DATA_BLOCK "Working_Programs"   // DB25
{ S7_Optimized_Access := 'FALSE' }
VERSION : 0.1
   VAR
      Count : USInt := 16;
      List : Array[0..21] of "RobotProgram";
   END_VAR
BEGIN
   List[4].Entry_Points[7].part_side := '';
   List[4].Entry_Points[7].operation_side := '';
   List[4].Entry_Points[7].lay_number := -1;
   List[4].Entry_Points[7].operation_type := 'transfer_slot2out';
   List[4].Entry_Points[7].part_destination := '';
   List[4].Entry_Points[7].part_status := 'gripper';
   List[4].Entry_Points[7].robot_status := 'home';
   List[4].Entry_Points[7].machine_status := '';
   List[4].Entry_Points[7].previous_trajectory := 'TakeFromSlot';
   List[4].Entry_Points[7].active := true;
   List[3].Entry_Points[3].part_side := '';
   List[3].Entry_Points[3].operation_side := '';
   List[3].Entry_Points[3].lay_number := -1;
   List[3].Entry_Points[3].operation_type := 'transfer_in2slot';
   List[3].Entry_Points[3].part_destination := 'part_slot';
   List[3].Entry_Points[3].part_status := 'gripper';
   List[3].Entry_Points[3].robot_status := 'pallet_in';
   List[3].Entry_Points[3].machine_status := '';
   List[3].Entry_Points[3].previous_trajectory := 'TakeFromPalletIn';
   List[3].Entry_Points[3].active := true;
   List[2].Entry_Points[1].operation_type := 'machining';
   List[2].Entry_Points[1].lay_number := -1;
   List[2].Entry_Points[1].operation_side := 'B';
   List[2].Entry_Points[1].part_side := 'B';
   List[2].Entry_Points[2].active := true;
   List[2].Entry_Points[2].previous_trajectory := 'AutoMachiningA_';
   List[2].Entry_Points[2].machine_status := '';
   List[2].Entry_Points[2].robot_status := 'flip_table';
   List[2].Entry_Points[2].part_status := 'flip_table';
   List[2].Entry_Points[2].part_destination := 'pallet_out';
   List[2].Entry_Points[2].operation_type := 'machining';
   List[2].Entry_Points[2].lay_number := -1;
   List[2].Entry_Points[2].operation_side := 'B';
   List[2].Entry_Points[2].part_side := 'B';
   List[15].Entry_Points[1].active := true;
   List[15].Entry_Points[1].previous_trajectory := 'Pallet_Scanning';
   List[15].Entry_Points[1].machine_status := '';
   List[15].Entry_Points[1].robot_status := 'home';
   List[15].Entry_Points[1].part_status := 'pallet_in';
   List[15].Entry_Points[1].part_destination := 'pallet_out';
   List[6].Entry_Points[9].part_side := 'A';
   List[6].Entry_Points[9].operation_side := 'A';
   List[6].Entry_Points[9].lay_number := -1;
   List[6].Entry_Points[9].operation_type := 'machining';
   List[6].Entry_Points[9].part_destination := '';
   List[6].Entry_Points[9].part_status := 'flip_table';
   List[6].Entry_Points[9].robot_status := 'flip_table';
   List[6].Entry_Points[9].machine_status := 'ready2load';
   List[6].Entry_Points[9].previous_trajectory := 'PutOnFlipTableB';
   List[6].Entry_Points[9].active := true;
   List[5].Entry_Points[4].part_side := 'B';
   List[5].Entry_Points[4].operation_side := 'B';
   List[5].Entry_Points[4].lay_number := -1;
   List[5].Entry_Points[4].operation_type := 'transfer_in2out';
   List[5].Entry_Points[4].part_destination := '';
   List[5].Entry_Points[4].part_status := 'gripper';
   List[5].Entry_Points[4].robot_status := 'pallet_in';
   List[5].Entry_Points[4].machine_status := '';
   List[5].Entry_Points[4].previous_trajectory := 'TakeFromPalletIn';
   List[5].Entry_Points[4].active := true;
   List[5].Entry_Points[3].part_side := 'B';
   List[5].Entry_Points[3].operation_side := 'B';
   List[5].Entry_Points[3].lay_number := -1;
   List[5].Entry_Points[3].operation_type := 'machining';
   List[5].Entry_Points[3].part_destination := '';
   List[5].Entry_Points[3].part_status := 'gripper';
   List[5].Entry_Points[3].robot_status := 'pallet_in';
   List[5].Entry_Points[3].machine_status := '';
   List[5].Entry_Points[3].previous_trajectory := 'TakeFromPalletIn';
   List[5].Entry_Points[3].active := true;
   List[4].Entry_Points[6].part_side := '';
   List[4].Entry_Points[6].operation_side := '';
   List[4].Entry_Points[6].lay_number := -1;
   List[4].Entry_Points[6].operation_type := 'transfer_in2out';
   List[4].Entry_Points[6].part_destination := '';
   List[4].Entry_Points[6].part_status := 'gripper';
   List[4].Entry_Points[6].robot_status := 'pallet_in';
   List[4].Entry_Points[6].machine_status := '';
   List[4].Entry_Points[6].previous_trajectory := 'AutoMachiningA_';
   List[4].Entry_Points[6].active := true;
   List[6].Entry_Points[8].part_side := '';
   List[6].Entry_Points[8].operation_side := '';
   List[6].Entry_Points[8].lay_number := -1;
   List[6].Entry_Points[8].operation_type := 'machining';
   List[6].Entry_Points[8].part_destination := '';
   List[6].Entry_Points[8].part_status := 'flip_table';
   List[6].Entry_Points[8].robot_status := 'home';
   List[6].Entry_Points[8].machine_status := '';
   List[6].Entry_Points[8].previous_trajectory := 'PutOnFlipTableA';
   List[6].Entry_Points[8].active := true;
   List[1].Entry_Points[4].part_side := '';
   List[1].Entry_Points[4].operation_side := '';
   List[1].Entry_Points[4].lay_number := -1;
   List[1].Entry_Points[4].operation_type := 'scanning';
   List[1].Entry_Points[4].part_destination := '';
   List[1].Entry_Points[4].part_status := '';
   List[1].Entry_Points[4].robot_status := 'flip_table';
   List[1].Entry_Points[4].machine_status := '';
   List[1].Entry_Points[4].previous_trajectory := '';
   List[1].Entry_Points[4].active := true;
   List[6].Entry_Points[7].active := true;
   List[6].Entry_Points[7].previous_trajectory := 'PutOnFlipTableB';
   List[6].Entry_Points[7].machine_status := 'ready2load';
   List[6].Entry_Points[7].robot_status := 'home';
   List[6].Entry_Points[7].part_status := 'flip_table';
   List[6].Entry_Points[7].part_destination := '';
   List[6].Entry_Points[7].operation_type := 'machining';
   List[6].Entry_Points[7].lay_number := -1;
   List[6].Entry_Points[7].operation_side := 'B';
   List[6].Entry_Points[7].part_side := 'B';
   List[10].Entry_Points[2].part_side := 'A';
   List[10].Entry_Points[2].operation_side := 'B';
   List[10].Entry_Points[2].lay_number := -1;
   List[10].Entry_Points[2].operation_type := 'machining';
   List[10].Entry_Points[2].part_destination := 'pallet_out';
   List[10].Entry_Points[2].part_status := 'gripper';
   List[10].Entry_Points[2].robot_status := 'pallet_in';
   List[10].Entry_Points[2].machine_status := '';
   List[10].Entry_Points[2].previous_trajectory := 'TakeFromPalletIn';
   List[10].Entry_Points[2].active := true;
   List[6].Entry_Points[6].part_side := 'B';
   List[6].Entry_Points[6].operation_side := 'B';
   List[6].Entry_Points[6].lay_number := -1;
   List[6].Entry_Points[6].operation_type := 'machining';
   List[13].trajectory := 'PutOnFlipTableB';
   List[13].Entry_Points[1].part_side := '';
   List[13].Entry_Points[1].operation_side := '';
   List[13].Entry_Points[1].lay_number := -1;
   List[13].Entry_Points[1].operation_type := 'machining';
   List[13].Entry_Points[1].part_destination := 'flip_table';
   List[13].Entry_Points[1].part_status := 'gripper';
   List[13].Entry_Points[1].robot_status := 'pallet_out';
   List[13].Entry_Points[1].machine_status := '';
   List[13].Entry_Points[1].previous_trajectory := 'UnloadMachine';
   List[13].Entry_Points[1].active := true;
   List[11].Entry_Points[1].part_side := '';
   List[11].Entry_Points[1].operation_side := '';
   List[11].Entry_Points[1].lay_number := -1;
   List[11].Entry_Points[1].operation_type := 'transfer_in2flip';
   List[11].Entry_Points[1].part_destination := '';
   List[11].Entry_Points[1].part_status := 'gripper';
   List[11].Entry_Points[1].robot_status := 'pallet_in';
   List[11].Entry_Points[1].machine_status := '';
   List[11].Entry_Points[1].previous_trajectory := 'TakeFromPalletIn';
   List[11].Entry_Points[1].active := true;
   List[7].Entry_Points[2].part_destination := '';
   List[6].Entry_Points[5].part_status := 'flip_table';
   List[6].Entry_Points[4].part_destination := '';
   List[5].Entry_Points[2].part_side := 'A';
   List[5].Entry_Points[2].operation_side := 'A';
   List[5].Entry_Points[2].lay_number := -1;
   List[5].Entry_Points[2].operation_type := 'machining';
   List[12].OUT_Status.inprocess_part_status := 'pallet_in';
   List[12].OUT_Status.finish_part_status := 'pallet_in';
   List[15].Entry_Points[1].operation_type := 'machining';
   List[15].Entry_Points[1].lay_number := -1;
   List[15].Entry_Points[1].operation_side := 'A';
   List[15].Entry_Points[1].part_side := 'A';
   List[15].Entry_Points[3].active := true;
   List[15].Entry_Points[3].previous_trajectory := 'PartHeightMeasuring';
   List[15].Entry_Points[3].machine_status := '';
   List[15].Entry_Points[3].robot_status := 'pallet_in';
   List[15].Entry_Points[3].part_status := 'pallet_in';
   List[15].Entry_Points[3].part_destination := 'pallet_out';
   List[9].Entry_Points[5].part_destination := '';
   List[9].Entry_Points[4].part_destination := '';
   List[15].Entry_Points[3].operation_type := 'machining';
   List[15].Entry_Points[3].lay_number := -1;
   List[15].Entry_Points[3].operation_side := 'A';
   List[15].Entry_Points[3].part_side := 'A';
   List[15].Entry_Points[2].active := true;
   List[15].Entry_Points[2].previous_trajectory := 'AutoMachiningA';
   List[15].Entry_Points[2].machine_status := '';
   List[15].Entry_Points[2].robot_status := 'flip_tabel';
   List[15].Entry_Points[2].part_status := 'pallet_in';
   List[15].Entry_Points[2].part_destination := 'pallet_out';
   List[15].Entry_Points[2].operation_type := 'machining';
   List[15].Entry_Points[2].lay_number := -1;
   List[15].Entry_Points[2].operation_side := 'A';
   List[15].Entry_Points[2].part_side := 'A';
   List[1].Entry_Points[3].part_side := '';
   List[1].Entry_Points[3].operation_side := '';
   List[1].Entry_Points[3].lay_number := -1;
   List[1].Entry_Points[3].operation_type := 'scanning';
   List[1].Entry_Points[3].part_destination := '';
   List[1].Entry_Points[3].part_status := '';
   List[1].Entry_Points[3].robot_status := 'pallet_out';
   List[1].Entry_Points[3].machine_status := '';
   List[1].Entry_Points[3].previous_trajectory := '';
   List[1].Entry_Points[3].active := true;
   List[12].Entry_Points[1].part_side := '';
   List[12].Entry_Points[1].operation_side := '';
   List[12].Entry_Points[1].lay_number := -1;
   List[12].Entry_Points[1].operation_type := 'go_home';
   List[12].Entry_Points[1].part_destination := '';
   List[12].Entry_Points[1].part_status := '';
   List[12].Entry_Points[1].machine_status := '';
   List[12].Entry_Points[1].previous_trajectory := '';
   List[12].Entry_Points[1].active := true;
   List[12].OUT_Status.finish_task_status := 'done';
   List[12].OUT_Status.inprocess_task_status := 'in_process';
   List[12].trajectory := 'go_home';
   List[9].Entry_Points[3].part_destination := '';
   List[1].Entry_Points[2].part_side := '';
   List[1].Entry_Points[2].operation_side := '';
   List[1].Entry_Points[2].lay_number := -1;
   List[1].Entry_Points[2].operation_type := 'scanning';
   List[1].Entry_Points[2].part_destination := '';
   List[1].Entry_Points[2].part_status := '';
   List[1].Entry_Points[2].robot_status := 'pallet_in';
   List[1].Entry_Points[2].machine_status := '';
   List[1].Entry_Points[2].previous_trajectory := '';
   List[1].Entry_Points[2].active := true;
   List[11].OUT_Status.finish_part_status := 'flip_table';
   List[11].OUT_Status.finish_task_status := 'done';
   List[11].OUT_Status.inprocess_part_status := 'dropping';
   List[11].OUT_Status.inprocess_task_status := 'in_process';
   List[10].Entry_Points[7].operation_side := '';
   List[10].Entry_Points[7].part_side := '';
   List[11].trajectory := 'PutOnFlipTableA';
   List[6].Entry_Points[2].part_destination := '';
   List[4].Entry_Points[2].part_destination := 'pallet_out';
   List[5].Entry_Points[1].part_destination := '';
   List[5].Entry_Points[2].active := true;
   List[11].Entry_Points[5].part_side := '';
   List[11].Entry_Points[5].operation_side := '';
   List[11].Entry_Points[5].lay_number := -1;
   List[11].Entry_Points[5].operation_type := '';
   List[11].Entry_Points[5].part_destination := '';
   List[11].Entry_Points[5].part_status := '';
   List[11].Entry_Points[5].robot_status := '';
   List[11].Entry_Points[5].machine_status := '';
   List[11].Entry_Points[5].previous_trajectory := '';
   List[11].Entry_Points[5].active := false;
   List[11].Entry_Points[4].part_side := '';
   List[11].Entry_Points[4].operation_side := '';
   List[11].Entry_Points[4].lay_number := -1;
   List[11].Entry_Points[4].operation_type := '';
   List[11].Entry_Points[4].part_destination := '';
   List[11].Entry_Points[4].part_status := '';
   List[11].Entry_Points[4].robot_status := '';
   List[11].Entry_Points[4].machine_status := '';
   List[11].Entry_Points[4].previous_trajectory := '';
   List[11].Entry_Points[4].active := false;
   List[11].Entry_Points[3].part_side := '';
   List[11].Entry_Points[3].operation_side := '';
   List[11].Entry_Points[3].lay_number := -1;
   List[11].Entry_Points[3].operation_type := '';
   List[11].Entry_Points[3].part_destination := '';
   List[11].Entry_Points[3].part_status := '';
   List[11].Entry_Points[3].robot_status := '';
   List[11].Entry_Points[3].machine_status := '';
   List[11].Entry_Points[3].previous_trajectory := '';
   List[11].Entry_Points[3].active := false;
   List[11].Entry_Points[2].part_side := ' ';
   List[11].Entry_Points[2].operation_side := ' ';
   List[11].Entry_Points[2].lay_number := -1;
   List[11].Entry_Points[2].operation_type := '';
   List[11].Entry_Points[2].part_destination := '';
   List[11].Entry_Points[2].part_status := '';
   List[11].Entry_Points[2].robot_status := '';
   List[11].Entry_Points[2].machine_status := '';
   List[11].Entry_Points[2].previous_trajectory := '';
   List[11].Entry_Points[2].active := false;
   List[10].OUT_Status.finish_part_status := 'flip_table';
   List[10].OUT_Status.finish_task_status := 'on_trajectory';
   List[10].OUT_Status.inprocess_part_status := 'dropping';
   List[10].OUT_Status.inprocess_task_status := 'in_process';
   List[10].Entry_Points[5].part_destination := '';
   List[10].Entry_Points[4].part_destination := 'pallet_out';
   List[10].Entry_Points[3].part_side := 'B';
   List[10].Entry_Points[3].operation_side := 'A';
   List[10].Entry_Points[3].lay_number := -1;
   List[10].Entry_Points[3].operation_type := 'machining';
   List[10].Entry_Points[3].part_destination := 'part_slot';
   List[10].Entry_Points[3].part_status := 'gripper';
   List[10].Entry_Points[3].robot_status := 'pallet_in';
   List[10].Entry_Points[3].machine_status := '';
   List[10].Entry_Points[3].previous_trajectory := 'TakeFromPalletIn';
   List[10].Entry_Points[3].active := true;
   List[13].OUT_Status.inprocess_task_status := 'in_process';
   List[13].OUT_Status.inprocess_part_status := 'dropping';
   List[13].OUT_Status.finish_task_status := 'done';
   List[13].OUT_Status.finish_part_status := 'flip_table';
   List[6].Entry_Points[6].active := true;
   List[6].Entry_Points[6].previous_trajectory := 'PutOnFlipTableB';
   List[6].Entry_Points[6].machine_status := 'ready2load';
   List[6].Entry_Points[6].robot_status := 'flip_table';
   List[6].Entry_Points[6].part_status := 'flip_table';
   List[6].Entry_Points[6].part_destination := '';
   List[10].Entry_Points[1].part_side := 'A';
   List[10].Entry_Points[1].operation_side := 'B';
   List[10].Entry_Points[1].lay_number := -1;
   List[10].Entry_Points[1].operation_type := 'machining';
   List[10].Entry_Points[1].part_destination := 'part_slot';
   List[10].Entry_Points[1].part_status := 'gripper';
   List[10].Entry_Points[1].robot_status := 'pallet_in';
   List[10].Entry_Points[1].machine_status := '';
   List[10].Entry_Points[1].previous_trajectory := 'TakeFromPalletIn';
   List[10].Entry_Points[1].active := true;
   List[10].trajectory := 'PutOnFlipTableB';
   List[3].Entry_Points[2].part_destination := 'part_slot';
   List[3].Entry_Points[1].part_destination := 'part_slot';
   List[10].Entry_Points[5].part_side := '';
   List[10].Entry_Points[5].operation_side := '';
   List[10].Entry_Points[5].lay_number := -1;
   List[10].Entry_Points[5].operation_type := '';
   List[10].Entry_Points[5].part_status := '';
   List[10].Entry_Points[5].robot_status := '';
   List[10].Entry_Points[5].machine_status := '';
   List[10].Entry_Points[5].previous_trajectory := '';
   List[10].Entry_Points[5].active := false;
   List[10].Entry_Points[4].part_side := 'B';
   List[10].Entry_Points[4].operation_side := 'A';
   List[10].Entry_Points[4].lay_number := -1;
   List[10].Entry_Points[4].operation_type := 'machining';
   List[10].Entry_Points[4].part_status := 'gripper';
   List[10].Entry_Points[4].robot_status := 'pallet_in';
   List[10].Entry_Points[4].machine_status := '';
   List[10].Entry_Points[4].previous_trajectory := 'TakeFromPalletIn';
   List[10].Entry_Points[4].active := true;
   List[3].Entry_Points[5].part_side := '';
   List[3].Entry_Points[5].operation_side := '';
   List[3].Entry_Points[5].lay_number := -1;
   List[3].Entry_Points[5].operation_type := '';
   List[3].Entry_Points[5].part_status := '';
   List[3].Entry_Points[5].robot_status := '';
   List[3].Entry_Points[5].machine_status := '';
   List[3].Entry_Points[5].previous_trajectory := '';
   List[3].Entry_Points[5].active := false;
   List[3].Entry_Points[4].part_side := '';
   List[3].Entry_Points[4].operation_side := '';
   List[3].Entry_Points[4].lay_number := -1;
   List[3].Entry_Points[4].operation_type := '';
   List[3].Entry_Points[4].part_status := '';
   List[3].Entry_Points[4].robot_status := '';
   List[3].Entry_Points[4].machine_status := '';
   List[3].Entry_Points[4].previous_trajectory := '';
   List[3].Entry_Points[4].active := false;
   List[9].Entry_Points[5].part_side := '';
   List[9].Entry_Points[5].operation_side := '';
   List[9].Entry_Points[5].lay_number := -1;
   List[9].Entry_Points[5].operation_type := 'machining';
   List[9].Entry_Points[5].part_status := 'part_slot';
   List[9].Entry_Points[5].robot_status := 'pallet_out';
   List[9].Entry_Points[5].machine_status := '';
   List[9].Entry_Points[5].previous_trajectory := '';
   List[9].Entry_Points[5].active := true;
   List[9].Entry_Points[4].part_side := '';
   List[9].Entry_Points[4].operation_side := '';
   List[9].Entry_Points[4].lay_number := -1;
   List[9].Entry_Points[4].operation_type := 'transfer_slot2out';
   List[9].Entry_Points[4].part_status := 'part_slot';
   List[9].Entry_Points[4].robot_status := 'pallet_out';
   List[9].Entry_Points[4].machine_status := '';
   List[9].Entry_Points[4].previous_trajectory := '';
   List[9].Entry_Points[4].active := true;
   List[9].Entry_Points[3].part_side := '';
   List[9].Entry_Points[3].operation_side := '';
   List[9].Entry_Points[3].lay_number := -1;
   List[9].Entry_Points[3].operation_type := 'transfer_slot2out';
   List[9].Entry_Points[3].part_status := 'part_slot';
   List[9].Entry_Points[3].robot_status := 'pallet_in';
   List[9].Entry_Points[3].machine_status := '';
   List[9].Entry_Points[3].previous_trajectory := '';
   List[9].Entry_Points[3].active := true;
   List[9].Entry_Points[2].part_side := '';
   List[9].Entry_Points[2].operation_side := '';
   List[9].Entry_Points[2].lay_number := -1;
   List[9].Entry_Points[2].operation_type := 'machining';
   List[9].Entry_Points[2].part_status := 'part_slot';
   List[9].Entry_Points[2].robot_status := 'home';
   List[9].Entry_Points[2].machine_status := '';
   List[9].Entry_Points[2].previous_trajectory := '';
   List[9].Entry_Points[2].active := true;
   List[9].Entry_Points[1].part_side := '';
   List[9].Entry_Points[1].operation_side := '';
   List[9].Entry_Points[1].lay_number := -1;
   List[9].Entry_Points[1].operation_type := 'transfer_slot2out';
   List[9].Entry_Points[1].part_status := 'part_slot';
   List[9].Entry_Points[1].robot_status := 'home';
   List[9].Entry_Points[1].machine_status := '';
   List[9].Entry_Points[1].previous_trajectory := '';
   List[9].Entry_Points[1].active := true;
   List[8].Entry_Points[5].part_side := '';
   List[8].Entry_Points[5].operation_side := '';
   List[8].Entry_Points[5].lay_number := -1;
   List[8].Entry_Points[5].operation_type := '';
   List[8].Entry_Points[5].part_status := '';
   List[8].Entry_Points[5].robot_status := '';
   List[8].Entry_Points[5].machine_status := '';
   List[8].Entry_Points[5].previous_trajectory := '';
   List[8].Entry_Points[5].active := false;
   List[8].Entry_Points[4].part_side := '';
   List[8].Entry_Points[4].operation_side := '';
   List[8].Entry_Points[4].lay_number := -1;
   List[8].Entry_Points[4].operation_type := '';
   List[8].Entry_Points[4].part_status := '';
   List[8].Entry_Points[4].robot_status := '';
   List[8].Entry_Points[4].machine_status := '';
   List[8].Entry_Points[4].previous_trajectory := '';
   List[8].Entry_Points[4].active := false;
   List[8].Entry_Points[3].part_side := '';
   List[8].Entry_Points[3].operation_side := '';
   List[8].Entry_Points[3].lay_number := -1;
   List[8].Entry_Points[3].operation_type := '';
   List[8].Entry_Points[3].part_status := '';
   List[8].Entry_Points[3].robot_status := '';
   List[8].Entry_Points[3].machine_status := '';
   List[8].Entry_Points[3].previous_trajectory := '';
   List[8].Entry_Points[3].active := false;
   List[8].Entry_Points[2].part_side := '';
   List[8].Entry_Points[2].operation_side := '';
   List[8].Entry_Points[2].machine_status := '';
   List[8].Entry_Points[1].part_side := '';
   List[8].Entry_Points[1].operation_side := '';
   List[8].Entry_Points[1].machine_status := 'ready2unload';
   List[1].Entry_Points[1].operation_type := 'scanning';
   List[7].Entry_Points[5].part_side := '';
   List[7].Entry_Points[5].operation_side := '';
   List[7].Entry_Points[5].lay_number := -1;
   List[7].Entry_Points[5].operation_type := '';
   List[7].Entry_Points[5].part_status := '';
   List[7].Entry_Points[5].robot_status := '';
   List[7].Entry_Points[5].machine_status := '';
   List[7].Entry_Points[5].previous_trajectory := '';
   List[7].Entry_Points[5].active := false;
   List[7].Entry_Points[3].part_side := '';
   List[7].Entry_Points[3].operation_side := '';
   List[7].Entry_Points[3].lay_number := -1;
   List[7].Entry_Points[3].operation_type := 'machining';
   List[7].Entry_Points[3].part_status := 'gripper';
   List[7].Entry_Points[3].robot_status := 'flip_table';
   List[7].Entry_Points[3].machine_status := 'ready2load';
   List[7].Entry_Points[3].previous_trajectory := 'TakeFromSlot';
   List[7].Entry_Points[3].active := true;
   List[7].Entry_Points[2].part_side := 'B';
   List[7].Entry_Points[2].operation_side := 'B';
   List[7].Entry_Points[2].lay_number := -1;
   List[7].Entry_Points[2].operation_type := 'machining';
   List[7].Entry_Points[2].part_status := 'gripper';
   List[7].Entry_Points[2].robot_status := 'flip_table';
   List[7].Entry_Points[2].machine_status := 'ready2load';
   List[7].Entry_Points[2].previous_trajectory := 'TakeFromFlipTabelA';
   List[7].Entry_Points[2].active := true;
   List[7].Entry_Points[1].part_side := 'A';
   List[7].Entry_Points[1].operation_side := 'A';
   List[7].Entry_Points[1].lay_number := -1;
   List[0].OUT_Status.finish_task_status := 'unknown';
   List[0].OUT_Status.finish_part_status := 'unknown';
   List[6].Entry_Points[5].active := true;
   List[6].Entry_Points[5].previous_trajectory := 'PutOnFlipTableA';
   List[6].Entry_Points[5].machine_status := 'ready2load';
   List[6].Entry_Points[5].robot_status := 'flip_table';
   List[6].Entry_Points[5].part_destination := '';
   List[6].Entry_Points[5].operation_type := 'machining';
   List[6].Entry_Points[5].lay_number := -1;
   List[6].Entry_Points[5].operation_side := 'B';
   List[6].Entry_Points[5].part_side := 'B';
   List[6].Entry_Points[4].part_side := '';
   List[6].Entry_Points[4].operation_side := '';
   List[6].Entry_Points[4].lay_number := -1;
   List[6].Entry_Points[4].operation_type := 'transfer_in2out';
   List[6].Entry_Points[4].part_status := 'flip_table';
   List[6].Entry_Points[4].robot_status := 'flip_table';
   List[6].Entry_Points[4].machine_status := '';
   List[6].Entry_Points[4].previous_trajectory := 'PutOnFlipTableA';
   List[6].Entry_Points[4].active := true;
   List[6].Entry_Points[3].part_side := '';
   List[6].Entry_Points[3].operation_side := '';
   List[6].Entry_Points[3].lay_number := -1;
   List[6].Entry_Points[3].operation_type := 'machining';
   List[6].Entry_Points[3].part_status := 'flip_table';
   List[6].Entry_Points[3].robot_status := 'flip_table';
   List[6].Entry_Points[3].machine_status := '';
   List[6].Entry_Points[3].previous_trajectory := 'PutOnFlipTableB';
   List[6].Entry_Points[3].active := true;
   List[6].Entry_Points[2].part_side := '';
   List[6].Entry_Points[2].operation_side := '';
   List[6].Entry_Points[2].lay_number := -1;
   List[6].Entry_Points[1].part_side := 'A';
   List[6].Entry_Points[1].operation_side := 'A';
   List[6].Entry_Points[1].lay_number := -1;
   List[5].Entry_Points[5].part_side := '';
   List[5].Entry_Points[5].operation_side := '';
   List[5].Entry_Points[5].lay_number := -1;
   List[5].Entry_Points[5].operation_type := '';
   List[5].Entry_Points[5].part_status := '';
   List[5].Entry_Points[5].robot_status := '';
   List[5].Entry_Points[5].machine_status := '';
   List[5].Entry_Points[5].previous_trajectory := '';
   List[5].Entry_Points[5].active := false;
   List[6].Entry_Points[3].part_destination := '';
   List[4].Entry_Points[4].part_destination := '';
   List[4].Entry_Points[5].part_destination := '';
   List[5].Entry_Points[2].previous_trajectory := 'TakeFromPalletIn';
   List[5].Entry_Points[2].machine_status := '';
   List[5].Entry_Points[2].robot_status := 'pallet_in';
   List[5].Entry_Points[2].part_status := 'gripper';
   List[5].Entry_Points[2].part_destination := '';
   List[5].Entry_Points[1].lay_number := -1;
   List[4].Entry_Points[5].part_side := '';
   List[4].Entry_Points[5].operation_side := '';
   List[4].Entry_Points[5].lay_number := -1;
   List[4].Entry_Points[5].operation_type := 'transfer_slot2out';
   List[4].Entry_Points[5].part_status := 'gripper';
   List[4].Entry_Points[5].robot_status := 'part_slot';
   List[4].Entry_Points[5].machine_status := '';
   List[4].Entry_Points[5].previous_trajectory := 'TakeFromSlot';
   List[4].Entry_Points[5].active := true;
   List[4].Entry_Points[4].part_side := '';
   List[4].Entry_Points[4].operation_side := '';
   List[4].Entry_Points[4].lay_number := -1;
   List[4].Entry_Points[4].operation_type := 'machining';
   List[4].Entry_Points[4].part_status := 'gripper';
   List[4].Entry_Points[4].robot_status := 'pallet_in';
   List[4].Entry_Points[4].machine_status := '';
   List[4].Entry_Points[4].previous_trajectory := 'PutOnPalletOut';
   List[4].Entry_Points[4].active := true;
   List[4].Entry_Points[3].part_side := '';
   List[4].Entry_Points[3].operation_side := '';
   List[4].Entry_Points[3].lay_number := -1;
   List[4].Entry_Points[3].operation_type := 'transfer_slot2out';
   List[4].Entry_Points[3].part_status := 'gripper';
   List[4].Entry_Points[3].robot_status := 'flip_table';
   List[4].Entry_Points[3].machine_status := '';
   List[4].Entry_Points[3].previous_trajectory := 'TakeFromSlot';
   List[4].Entry_Points[3].active := true;
   List[4].Entry_Points[2].part_side := '';
   List[4].Entry_Points[2].operation_side := '';
   List[4].Entry_Points[2].lay_number := -1;
   List[4].Entry_Points[2].operation_type := 'machining';
   List[4].Entry_Points[2].part_status := 'gripper';
   List[4].Entry_Points[2].robot_status := 'pallet_out';
   List[4].Entry_Points[2].machine_status := '';
   List[4].Entry_Points[2].previous_trajectory := 'UnloadMachine';
   List[4].Entry_Points[2].active := true;
   List[4].Entry_Points[1].lay_number := -1;
   List[8].Entry_Points[2].part_status := '';
   List[8].Entry_Points[2].robot_status := '';
   List[8].Entry_Points[1].part_status := 'in_machine';
   List[8].Entry_Points[1].previous_trajectory := 'LoadMachine';
   List[8].Entry_Points[1].operation_type := 'machining';
   List[8].Entry_Points[1].lay_number := -1;
   List[8].Entry_Points[1].active := true;
   List[8].Entry_Points[2].lay_number := -1;
   List[8].Entry_Points[2].operation_type := '';
   List[8].Entry_Points[2].active := false;
   List[7].Entry_Points[1].part_status := 'gripper';
   List[7].Entry_Points[1].robot_status := 'flip_table';
   List[7].Entry_Points[1].machine_status := 'ready2load';
   List[7].Entry_Points[1].previous_trajectory := 'TakeFromFlipTabelA';
   List[7].Entry_Points[1].active := true;
   List[7].Entry_Points[1].operation_type := 'machining';
   List[6].Entry_Points[1].operation_type := 'machining';
   List[6].Entry_Points[2].operation_type := 'machining';
   List[6].Entry_Points[2].previous_trajectory := 'PutOnFlipTableA';
   List[6].Entry_Points[1].previous_trajectory := 'PutOnFlipTableA';
   List[6].Entry_Points[2].part_status := 'flip_table';
   List[6].Entry_Points[2].robot_status := 'flip_table';
   List[6].Entry_Points[2].machine_status := '';
   List[6].Entry_Points[1].part_status := 'flip_table';
   List[6].Entry_Points[1].robot_status := 'flip_table';
   List[6].Entry_Points[1].machine_status := 'ready2load';
   List[6].Entry_Points[2].active := true;
   List[6].Entry_Points[1].active := true;
   List[4].Entry_Points[1].operation_type := 'transfer_in2out';
   List[5].Entry_Points[1].operation_type := 'transfer_in2out';
   List[5].Entry_Points[1].part_status := 'gripper';
   List[5].Entry_Points[1].robot_status := 'pallet_in';
   List[5].Entry_Points[1].machine_status := '';
   List[5].Entry_Points[1].part_side := 'A';
   List[5].Entry_Points[1].operation_side := 'A';
   List[5].Entry_Points[1].previous_trajectory := 'TakeFromPalletIn';
   List[6].OUT_Status.finish_part_status := 'gripper';
   List[6].OUT_Status.finish_task_status := 'on_trajectory';
   List[6].OUT_Status.inprocess_part_status := 'flipping';
   List[6].OUT_Status.inprocess_task_status := 'in_process';
   List[8].Entry_Points[2].previous_trajectory := '';
   List[5].OUT_Status.finish_part_status := 'flip_table';
   List[5].OUT_Status.finish_task_status := 'on_trajectory';
   List[5].OUT_Status.inprocess_part_status := 'dropping';
   List[5].OUT_Status.inprocess_task_status := 'in_process';
   List[4].OUT_Status.finish_part_status := 'pallet_out';
   List[4].OUT_Status.finish_task_status := 'done';
   List[4].OUT_Status.inprocess_part_status := 'dropping';
   List[4].OUT_Status.inprocess_task_status := 'in_process';
   List[4].trajectory := 'PutOnPalletOut';
   List[3].Entry_Points[1].lay_number := -1;
   List[8].Entry_Points[1].robot_status := 'at_machine';
   List[3].Entry_Points[1].machine_status := '';
   List[3].Entry_Points[1].operation_side := '';
   List[3].Entry_Points[1].part_side := '';
   List[3].Entry_Points[2].lay_number := -1;
   List[3].Entry_Points[2].machine_status := '';
   List[3].Entry_Points[2].previous_trajectory := 'UnloadMachine';
   List[3].Entry_Points[2].active := true;
   List[9].trajectory := 'TakeFromSlot';
   List[3].Entry_Points[1].active := true;
   List[3].Entry_Points[2].part_side := '';
   List[3].Entry_Points[1].robot_status := 'flip_table';
   List[4].Entry_Points[1].machine_status := '';
   List[4].Entry_Points[1].robot_status := 'flip_table';
   List[4].Entry_Points[1].part_status := 'gripper';
   List[4].Entry_Points[1].previous_trajectory := 'TakeFromFlipTabelA';
   List[4].Entry_Points[1].active := true;
   List[4].Entry_Points[1].operation_side := '';
   List[4].Entry_Points[1].part_side := '';
   List[5].Entry_Points[1].active := true;
   List[5].trajectory := 'PutOnFlipTableA';
   List[3].Entry_Points[2].part_status := 'gripper';
   List[9].OUT_Status.inprocess_part_status := 'grabbing';
   List[9].OUT_Status.finish_part_status := 'gripper';
   List[3].Entry_Points[1].operation_type := 'transfer_in2out';
   List[8].OUT_Status.finish_task_status := 'on_trajectory';
   List[8].OUT_Status.inprocess_task_status := 'in_process';
   List[7].OUT_Status.finish_task_status := 'on_trajectory';
   List[7].OUT_Status.inprocess_task_status := 'in_process';
   List[3].OUT_Status.finish_task_status := 'done';
   List[3].OUT_Status.inprocess_task_status := 'in_process';
   List[1].OUT_Status.finish_task_status := 'done';
   List[1].OUT_Status.inprocess_task_status := 'in_process';
   List[9].OUT_Status.finish_task_status := 'on_trajectory';
   List[3].Entry_Points[2].robot_status := 'pallet_out';
   List[8].OUT_Status.inprocess_part_status := 'unloading';
   List[7].OUT_Status.inprocess_part_status := 'loading';
   List[1].OUT_Status.inprocess_part_status := 'pallet_in';
   List[1].Entry_Points[1].robot_status := 'home';
   List[9].OUT_Status.inprocess_task_status := 'in_process';
   List[1].Entry_Points[1].active := true;
   List[3].Entry_Points[1].previous_trajectory := 'TakeFromFlipTabelA';
   List[3].Entry_Points[2].operation_side := '';
   List[3].Entry_Points[1].part_status := 'gripper';
   List[3].Entry_Points[2].operation_type := 'machining';
   List[8].trajectory := 'UnloadMachine';
   List[3].OUT_Status.inprocess_part_status := 'dropping';
   List[8].OUT_Status.finish_part_status := 'gripper';
   List[7].trajectory := 'LoadMachine';
   List[7].OUT_Status.finish_part_status := 'in_machine';
   List[6].trajectory := 'TakeFromFlipTableA';
   List[3].trajectory := 'PutOnSlot';
   List[3].OUT_Status.finish_part_status := 'part_slot';
   List[2].trajectory := 'AutoMachining_B';
   List[1].trajectory := 'Scanning';
   List[1].OUT_Status.finish_part_status := 'pallet_in';
   List[2].Entry_Points[1].part_destination := 'pallet_out';
   List[2].Entry_Points[1].part_status := 'flip_table';
   List[2].Entry_Points[1].robot_status := 'flip_table';
   List[2].Entry_Points[1].machine_status := '';
   List[2].Entry_Points[1].previous_trajectory := 'PutOnFlipTableB';
   List[2].Entry_Points[1].active := true;
   List[15].OUT_Status.finish_part_status := 'pallet_out';
   List[15].OUT_Status.inprocess_part_status := 'machining';
   List[15].OUT_Status.inprocess_task_status := 'in_process';
   List[15].OUT_Status.finish_task_status := 'done';
   List[14].trajectory := 'PartHeightMeasuring';
   List[14].Entry_Points[1].operation_type := 'measuring_height';
   List[14].Entry_Points[1].active := true;
   List[14].Entry_Points[2].operation_type := 'measuring_height';
   List[14].Entry_Points[2].active := true;
   List[14].Entry_Points[1].previous_trajectory := '';
   List[14].Entry_Points[2].previous_trajectory := 'PartHeightMeasuring';
   List[14].Entry_Points[1].robot_status := 'home';
   List[14].Entry_Points[2].robot_status := '';
   List[14].Entry_Points[2].part_status := 'scanned';
   List[14].Entry_Points[1].part_status := 'scanned';
   List[14].OUT_Status.inprocess_task_status := 'in_process';
   List[14].OUT_Status.inprocess_part_status := 'measuring';
   List[14].OUT_Status.finish_task_status := 'done';
   List[14].OUT_Status.finish_part_status := 'pallet_in';
   List[14].Entry_Points[3].active := true;
   List[14].Entry_Points[3].previous_trajectory := 'PartHeightMeasuring';
   List[14].Entry_Points[3].machine_status := '';
   List[14].Entry_Points[3].robot_status := '';
   List[14].Entry_Points[3].part_status := 'ordered';
   List[14].Entry_Points[3].part_destination := '';
   List[14].Entry_Points[3].operation_type := 'measuring_height';
   List[14].Entry_Points[4].part_status := 'pallet_in';
   List[14].Entry_Points[4].operation_type := 'measuring_height';
   List[14].Entry_Points[4].active := true;
   List[17].OUT_Status.inprocess_task_status := 'in_process';
   List[17].OUT_Status.inprocess_part_status := 'machining';
   List[17].OUT_Status.finish_task_status := 'done';
   List[17].OUT_Status.finish_part_status := 'flip_table';
   List[17].trajectory := 'AutoMachiningA_';
   List[17].Entry_Points[1].active := true;
   List[17].Entry_Points[1].previous_trajectory := 'Pallet_Scanning';
   List[17].Entry_Points[1].machine_status := '';
   List[17].Entry_Points[1].robot_status := 'pallet_in';
   List[17].Entry_Points[1].part_status := 'pallet_in';
   List[17].Entry_Points[1].part_destination := 'flip_table';
   List[17].Entry_Points[1].operation_type := 'machining';
   List[17].Entry_Points[1].lay_number := -1;
   List[17].Entry_Points[1].operation_side := 'A';
   List[17].Entry_Points[1].part_side := 'A';
   List[17].Entry_Points[2].active := true;
   List[17].Entry_Points[2].previous_trajectory := 'PutOnPalletOut';
   List[17].Entry_Points[2].machine_status := '';
   List[17].Entry_Points[2].robot_status := 'pallet_in';
   List[17].Entry_Points[2].part_status := 'pallet_in';
   List[17].Entry_Points[2].part_destination := 'flip_table';
   List[17].Entry_Points[2].operation_type := 'machining';
   List[17].Entry_Points[2].lay_number := -1;
   List[17].Entry_Points[2].operation_side := 'A';
   List[17].Entry_Points[2].part_side := 'A';
   List[16].Entry_Points[4].active := false;
   List[16].Entry_Points[4].previous_trajectory := '';
   List[16].Entry_Points[4].machine_status := '';
   List[16].Entry_Points[4].robot_status := '';
   List[16].Entry_Points[4].part_status := '';
   List[16].Entry_Points[4].part_destination := '';
   List[16].Entry_Points[4].operation_type := '';
   List[16].Entry_Points[4].lay_number := -1;
   List[16].Entry_Points[4].operation_side := '';
   List[16].Entry_Points[4].part_side := '';
   List[17].Entry_Points[3].active := true;
   List[17].Entry_Points[3].previous_trajectory := 'AutoMachiningB';
   List[17].Entry_Points[3].machine_status := '';
   List[17].Entry_Points[3].robot_status := 'pallet_in';
   List[17].Entry_Points[3].part_status := 'pallet_in';
   List[17].Entry_Points[3].part_destination := 'flip_table';
   List[17].Entry_Points[3].operation_type := 'machining';
   List[17].Entry_Points[3].lay_number := -1;
   List[17].Entry_Points[3].operation_side := 'A';
   List[17].Entry_Points[3].part_side := 'A';
   List[17].Entry_Points[4].active := true;
   List[17].Entry_Points[4].previous_trajectory := 'PartHeightMeasuring';
   List[17].Entry_Points[4].machine_status := '';
   List[17].Entry_Points[4].robot_status := 'pallet_in';
   List[17].Entry_Points[4].part_status := 'pallet_in';
   List[17].Entry_Points[4].part_destination := 'flip_table';
   List[17].Entry_Points[4].operation_type := 'machining';
   List[17].Entry_Points[4].lay_number := -1;
   List[17].Entry_Points[4].operation_side := 'A';
   List[17].Entry_Points[4].part_side := 'A';
   List[15].Entry_Points[4].active := true;
   List[15].Entry_Points[4].previous_trajectory := 'AutoMachiningB';
   List[15].Entry_Points[4].machine_status := '';
   List[15].Entry_Points[4].robot_status := 'flip_tabel';
   List[15].Entry_Points[4].part_status := 'pallet_in';
   List[15].Entry_Points[4].part_destination := 'pallet_out';
   List[15].Entry_Points[4].operation_type := 'machining';
   List[15].Entry_Points[4].lay_number := -1;
   List[15].Entry_Points[4].operation_side := 'A';
   List[15].Entry_Points[4].part_side := 'A';
   List[15].Entry_Points[5].active := true;
   List[15].Entry_Points[5].previous_trajectory := 'AutoMachining_B';
   List[15].Entry_Points[5].machine_status := '';
   List[15].Entry_Points[5].robot_status := 'flip_tabel';
   List[15].Entry_Points[5].part_status := 'pallet_in';
   List[15].Entry_Points[5].part_destination := 'pallet_out';
   List[15].Entry_Points[5].operation_type := 'machining';
   List[15].Entry_Points[5].lay_number := -1;
   List[15].Entry_Points[5].operation_side := 'A';
   List[15].Entry_Points[5].part_side := 'A';
   List[15].trajectory := 'AutoMachiningA';
   List[16].OUT_Status.inprocess_task_status := 'in_process';
   List[16].OUT_Status.inprocess_part_status := 'machining';
   List[16].OUT_Status.finish_task_status := 'done';
   List[16].OUT_Status.finish_part_status := 'pallet_out';
   List[16].trajectory := 'AutoMachiningB';
   List[16].Entry_Points[1].active := true;
   List[16].Entry_Points[1].previous_trajectory := 'AutoMachiningA';
   List[16].Entry_Points[1].machine_status := '';
   List[16].Entry_Points[1].robot_status := 'flip_table';
   List[16].Entry_Points[1].part_status := 'pallet_in';
   List[16].Entry_Points[1].part_destination := 'pallet_out';
   List[16].Entry_Points[1].operation_type := 'machining';
   List[16].Entry_Points[1].lay_number := -1;
   List[16].Entry_Points[1].operation_side := 'B';
   List[16].Entry_Points[1].part_side := 'A';
   List[16].Entry_Points[2].active := true;
   List[16].Entry_Points[2].previous_trajectory := 'AutoMachiningB';
   List[16].Entry_Points[2].machine_status := '';
   List[16].Entry_Points[2].robot_status := 'flip_table';
   List[16].Entry_Points[2].part_status := 'pallet_in';
   List[16].Entry_Points[2].part_destination := 'pallet_out';
   List[16].Entry_Points[2].operation_type := 'machining';
   List[16].Entry_Points[2].lay_number := -1;
   List[16].Entry_Points[2].operation_side := 'B';
   List[16].Entry_Points[2].part_side := 'A';
   List[16].Entry_Points[3].active := true;
   List[16].Entry_Points[3].previous_trajectory := 'AutoMachining_B';
   List[16].Entry_Points[3].machine_status := '';
   List[16].Entry_Points[3].robot_status := 'flip_table';
   List[16].Entry_Points[3].part_status := 'pallet_in';
   List[16].Entry_Points[3].part_destination := 'pallet_out';
   List[16].Entry_Points[3].operation_type := 'machining';
   List[16].Entry_Points[3].lay_number := -1;
   List[16].Entry_Points[3].operation_side := 'B';
   List[16].Entry_Points[3].part_side := 'A';
   List[18].trajectory := 'TakeFromPalletIn';
   List[18].Entry_Points[1].active := true;
   List[18].Entry_Points[1].previous_trajectory := '';
   List[18].Entry_Points[1].machine_status := 'ready2load';
   List[18].Entry_Points[1].robot_status := 'home';
   List[18].Entry_Points[1].part_status := 'pallet_in';
   List[18].Entry_Points[1].part_destination := '';
   List[18].Entry_Points[1].operation_type := 'machining';
   List[18].Entry_Points[1].lay_number := -1;
   List[18].Entry_Points[1].operation_side := '';
   List[18].Entry_Points[1].part_side := '';
   List[18].Entry_Points[2].active := true;
   List[18].Entry_Points[2].previous_trajectory := '';
   List[18].Entry_Points[2].machine_status := '';
   List[18].Entry_Points[2].robot_status := 'home';
   List[18].Entry_Points[2].part_status := 'pallet_in';
   List[18].Entry_Points[2].part_destination := '';
   List[18].Entry_Points[2].operation_type := 'transfer_in2out';
   List[18].Entry_Points[2].lay_number := -1;
   List[18].Entry_Points[2].operation_side := '';
   List[18].Entry_Points[2].part_side := '';
   List[18].Entry_Points[3].active := true;
   List[18].Entry_Points[3].previous_trajectory := '';
   List[18].Entry_Points[3].machine_status := '';
   List[18].Entry_Points[3].robot_status := 'home';
   List[18].Entry_Points[3].part_status := 'pallet_in';
   List[18].Entry_Points[3].part_destination := '';
   List[18].Entry_Points[3].operation_type := 'transfer_in2flip';
   List[18].Entry_Points[3].lay_number := -1;
   List[18].Entry_Points[3].operation_side := '';
   List[18].Entry_Points[3].part_side := '';
   List[18].Entry_Points[4].active := true;
   List[18].Entry_Points[4].previous_trajectory := '';
   List[18].Entry_Points[4].machine_status := 'ready2load';
   List[18].Entry_Points[4].robot_status := 'pallet_in';
   List[18].Entry_Points[4].part_status := 'pallet_in';
   List[18].Entry_Points[4].part_destination := '';
   List[18].Entry_Points[4].operation_type := 'machining';
   List[18].Entry_Points[4].lay_number := -1;
   List[18].Entry_Points[4].operation_side := '';
   List[18].Entry_Points[4].part_side := '';
   List[18].Entry_Points[5].active := true;
   List[18].Entry_Points[5].previous_trajectory := '';
   List[18].Entry_Points[5].machine_status := '';
   List[18].Entry_Points[5].robot_status := 'pallet_in';
   List[18].Entry_Points[5].part_status := 'pallet_in';
   List[18].Entry_Points[5].part_destination := '';
   List[18].Entry_Points[5].operation_type := 'transfer_in2flip';
   List[18].Entry_Points[5].lay_number := -1;
   List[18].Entry_Points[5].operation_side := '';
   List[18].Entry_Points[5].part_side := '';
   List[18].Entry_Points[6].active := true;
   List[18].Entry_Points[6].previous_trajectory := '';
   List[18].Entry_Points[6].machine_status := 'ready2load';
   List[18].Entry_Points[6].robot_status := 'pallet_out';
   List[18].Entry_Points[6].part_status := 'pallet_in';
   List[18].Entry_Points[6].part_destination := '';
   List[18].Entry_Points[6].operation_type := 'machining';
   List[18].Entry_Points[6].lay_number := -1;
   List[18].Entry_Points[6].operation_side := '';
   List[18].Entry_Points[6].part_side := '';
   List[18].Entry_Points[7].active := true;
   List[18].Entry_Points[7].previous_trajectory := '';
   List[18].Entry_Points[7].machine_status := '';
   List[18].Entry_Points[7].robot_status := 'pallet_out';
   List[18].Entry_Points[7].part_status := 'pallet_in';
   List[18].Entry_Points[7].part_destination := '';
   List[18].Entry_Points[7].operation_type := 'transfer_in2out';
   List[18].Entry_Points[7].lay_number := -1;
   List[18].Entry_Points[7].operation_side := '';
   List[18].Entry_Points[7].part_side := '';
   List[18].Entry_Points[8].active := true;
   List[18].Entry_Points[8].previous_trajectory := '';
   List[18].Entry_Points[8].machine_status := '';
   List[18].Entry_Points[8].robot_status := 'pallet_out';
   List[18].Entry_Points[8].part_status := 'pallet_in';
   List[18].Entry_Points[8].part_destination := '';
   List[18].Entry_Points[8].operation_type := 'transfer_in2flip';
   List[18].Entry_Points[8].lay_number := -1;
   List[18].Entry_Points[8].operation_side := '';
   List[18].Entry_Points[8].part_side := '';
   List[18].Entry_Points[9].active := true;
   List[18].Entry_Points[9].previous_trajectory := '';
   List[18].Entry_Points[9].machine_status := 'ready2load';
   List[18].Entry_Points[9].robot_status := 'flip_table';
   List[18].Entry_Points[9].part_status := 'pallet_in';
   List[18].Entry_Points[9].part_destination := '';
   List[18].Entry_Points[9].operation_type := 'machining';
   List[18].Entry_Points[9].lay_number := -1;
   List[18].Entry_Points[9].operation_side := '';
   List[18].Entry_Points[9].part_side := '';
   List[18].Entry_Points[10].active := true;
   List[18].Entry_Points[10].previous_trajectory := '';
   List[18].Entry_Points[10].machine_status := '';
   List[18].Entry_Points[10].robot_status := 'home';
   List[18].Entry_Points[10].part_status := 'pallet_in';
   List[18].Entry_Points[10].part_destination := '';
   List[18].Entry_Points[10].operation_type := 'transfer_in2slot';
   List[18].Entry_Points[10].lay_number := -1;
   List[18].Entry_Points[10].operation_side := '';
   List[18].Entry_Points[10].part_side := '';
   List[18].Entry_Points[11].active := true;
   List[18].Entry_Points[11].previous_trajectory := '';
   List[18].Entry_Points[11].machine_status := '';
   List[18].Entry_Points[11].robot_status := 'pallet_in';
   List[18].Entry_Points[11].part_status := 'pallet_in';
   List[18].Entry_Points[11].part_destination := '';
   List[18].Entry_Points[11].operation_type := 'transfer_in2slot';
   List[18].Entry_Points[11].lay_number := -1;
   List[18].Entry_Points[11].operation_side := '';
   List[18].Entry_Points[11].part_side := '';
   List[18].Entry_Points[12].active := true;
   List[18].Entry_Points[12].previous_trajectory := '';
   List[18].Entry_Points[12].machine_status := '';
   List[18].Entry_Points[12].robot_status := 'flip_table';
   List[18].Entry_Points[12].part_status := 'pallet_in';
   List[18].Entry_Points[12].part_destination := '';
   List[18].Entry_Points[12].operation_type := 'transfer_in2flip';
   List[18].Entry_Points[12].lay_number := -1;
   List[18].Entry_Points[12].operation_side := '';
   List[18].Entry_Points[12].part_side := '';
   List[18].OUT_Status.inprocess_task_status := 'in_process';
   List[18].OUT_Status.inprocess_part_status := 'grabbing';
   List[18].OUT_Status.finish_task_status := 'on_trajectory';
   List[18].OUT_Status.finish_part_status := 'gripper';
   List[2].OUT_Status.inprocess_task_status := 'in_process';
   List[2].OUT_Status.inprocess_part_status := 'machining';
   List[2].OUT_Status.finish_task_status := 'done';
   List[2].OUT_Status.finish_part_status := 'pallet_out';
END_DATA_BLOCK

// folder: 5_Matrix_scanner

DATA_BLOCK "DADProtocol_DB"   // DB6
{ S7_Optimized_Access := 'TRUE' }
VERSION : 0.1
// stored: InstanceOfName DADProtocol
"DADProtocol"
BEGIN
END_DATA_BLOCK

DATA_BLOCK "Matrix_output"   // DB10
{ S7_Optimized_Access := 'FALSE' }
VERSION : 0.1
   VAR
      new_code : Bool;
      scan_robot_pos_X : Real;
      scan_robot_pos_Y : Real;
      scan_robot_pos_Z : Real;
      scan_robot_angle_A : Real;
      scan_lay_number : USInt := 2;
      QR_codes_DAD : Array[0..512] of Byte;
   END_VAR
BEGIN
END_DATA_BLOCK

DATA_BLOCK "Timer_ON"   // DB11
{ S7_Optimized_Access := 'TRUE' }
AUTHOR : Simatic
FAMILY : IEC
NAME : IEC_TMR
VERSION : 1.0
// stored: InstanceOfName IEC_TIMER
"IEC_TIMER"
BEGIN
END_DATA_BLOCK

DATA_BLOCK "Timer_OFF"   // DB12
{ S7_Optimized_Access := 'TRUE' }
AUTHOR : Simatic
FAMILY : IEC
NAME : IEC_TMR
VERSION : 1.0
// stored: InstanceOfName IEC_TIMER
"IEC_TIMER"
BEGIN
END_DATA_BLOCK

DATA_BLOCK "Matrix_reading"   // DB14
{ S7_Optimized_Access := 'FALSE' }
VERSION : 0.1
   VAR
      new_code_readed : Bool;
      code_trigger : Bool;
      code_memory : Bool;
      last_code_ok : Bool;
      code_reading_ok : Bool;
      dad_enable : Bool;
      inputArrayCHARS : Array[0..62] of Char;
      pointerCHARS : DInt;
      countCHARS : UInt;
      QR_codes : String;
   END_VAR
BEGIN
END_DATA_BLOCK

// folder: 6_OPC

DATA_BLOCK "RobotTasks"   // DB1
{ S7_Optimized_Access := 'FALSE' }
VERSION : 0.1
   VAR
      Robot1 : "TypeRobotTask";
   END_VAR
BEGIN
END_DATA_BLOCK

DATA_BLOCK "WorkingTasks"   // DB5
{ S7_Optimized_Access := 'FALSE' }
VERSION : 0.1
   VAR
      Robot1 : "TypeRobotTask";
   END_VAR
BEGIN
END_DATA_BLOCK

DATA_BLOCK "Timers"   // DB18
{ S7_Optimized_Access := 'TRUE' }
VERSION : 0.1
   VAR
      button_Start_R : Bool;
      button_Reset_R : Bool;
   END_VAR
BEGIN
END_DATA_BLOCK

DATA_BLOCK "Pallet"   // DB20
{ S7_Optimized_Access := 'FALSE' }
VERSION : 0.1
   VAR
      new_label : Bool;
      pallet_pos_X : Int := 0;
      pallet_pos_Y : Int := 0;
      pallet_pos_Z : Int := 0;
      pallet_angle_A : Int;
   END_VAR
BEGIN
END_DATA_BLOCK

DATA_BLOCK "Robot"   // DB21
{ S7_Optimized_Access := 'FALSE' }
VERSION : 0.1
   VAR
      ALARM_STOP_KRC : Bool;
      EXT_ACTIVE : Bool;
      PERI_RDY_KRC : Bool;
      STOPMESS_KRC : Bool;
      IN_HOME_KRC : Bool;
      PRO_MOVE_KRC : Bool;
      PGNO_REFL_KRC : UInt;
      PGNO_REQ_KRC : Bool;
      USER_SAF_KRC : Bool;
      ROB_CAL_KRC : Bool;
      I_O_ACTCONF_KRC : Bool;
      RC_RDY1_KRC : Bool;
      APPL_RUN_KRC : Bool;
      Cam : Bool;
      LifeBit : Bool;
      EXT_FIRST_START : Bool;
      SetVacuumON : Bool;
      SetPressureOFF : Bool;
      SetRetract : Bool;
      Flow2PartON : Bool;
      SetFlipClose : Bool;
      PartOK : Bool;
      PartMeasuring : Bool;
      PRO_ACT_KRC : Bool;
      ERROR_KRC : Bool;
      AXIS_ACT_A1 : Real;
      POS_ACT_Z : Real;
      POS_ACT_Y : Real;
      POS_ACT_X : Real;
      POS_ACT_A : Real;
      Pallet_Scanned : Bool;
      FlipVacuumOn : Bool;
      Part_Status : UInt;
      Serial_Number : UInt;
   END_VAR
BEGIN
END_DATA_BLOCK

// folder: 7_Tags

DATA_BLOCK "PLC_tags"   // DB1000
{ S7_Optimized_Access := 'FALSE' }
VERSION : 0.1
   VAR
      Tags_count : Int := 0;
      Tags : Array[0..101] of "PLC_Tag";
   END_VAR
BEGIN
END_DATA_BLOCK

// folder: System blocks/Program resources

DATA_BLOCK "Pallet_start_timer"   // DB9
{ S7_Optimized_Access := 'TRUE' }
AUTHOR : Simatic
FAMILY : IEC
NAME : IEC_TMR
VERSION : 1.0
// stored: InstanceOfName IEC_TIMER
"IEC_TIMER"
BEGIN
END_DATA_BLOCK

DATA_BLOCK "Go_home_timer"   // DB16
{ S7_Optimized_Access := 'TRUE' }
AUTHOR : Simatic
FAMILY : IEC
NAME : IEC_TMR
VERSION : 1.0
// stored: InstanceOfName IEC_TIMER
"IEC_TIMER"
BEGIN
END_DATA_BLOCK

// folder: (top level)

FUNCTION_BLOCK "Default_SupervisionFB"   // FB1, ProDiag
{ S7_Optimized_Access := 'TRUE' }
   VAR
      PC_Flags : PC_Flags_V2;
      State : SV_FB_State_V2;
   END_VAR
   VAR_TEMP
      t_TempSvStateUDT : SV_State_V2;
      t_TempAlarmInstance : <type 200004f>;
      t_TempAsocValue1 : Variant;
      t_TempAsocValue2 : Variant;
      t_TempAsocValue3 : Variant;
   END_VAR
BEGIN
END_FUNCTION_BLOCK

ORGANIZATION_BLOCK "Main"   // OB1, LAD, ProgramCycle
TITLE = "Main Program Sweep (Cycle)"
{ S7_Optimized_Access := 'TRUE' }
VERSION : 0.1
   VAR_INPUT
      Initial_Call : Bool;   // Initial call of this OB
      Remanence : Bool;   // =True, if remanent data are available
   END_VAR
   VAR_TEMP
      Alarm_reset : Bool;
      Alarms_out : Bool;
   END_VAR
BEGIN

REGION Network 1
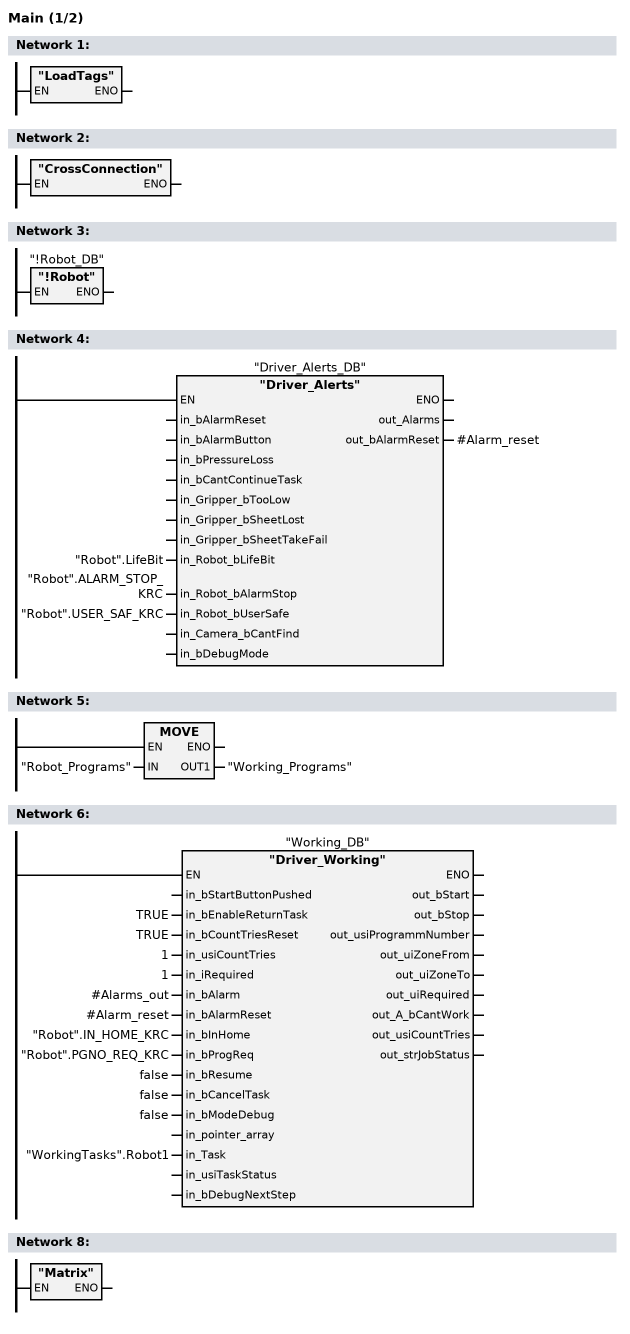
   RUNG wire#powerrail
      "LoadTags"()
   END_RUNG
   // the same network as SCL:
   "LoadTags"();
END_REGION

REGION Network 2
   RUNG wire#powerrail
      "CrossConnection"()
   END_RUNG
   // the same network as SCL:
   "CrossConnection"();
END_REGION

REGION Network 3
   RUNG wire#powerrail
      "!Robot_DB"()
   END_RUNG
   // the same network as SCL:
   "!Robot_DB"();   // "!Robot"
END_REGION

REGION Network 4
   RUNG wire#powerrail
      "Driver_Alerts_DB"(in_bAlarmReset :=, in_bAlarmButton :=, in_bPressureLoss :=, in_bCantContinueTask :=, in_Gripper_bTooLow :=, in_Gripper_bSheetLost :=, in_Gripper_bSheetTakeFail :=, in_Robot_bLifeBit := "Robot".LifeBit, in_Robot_bAlarmStop := "Robot".ALARM_STOP_KRC, in_Robot_bUserSafe := "Robot".USER_SAF_KRC, in_Camera_bCantFind :=, in_bDebugMode :=, out_Alarms =>, out_bAlarmReset => #Alarm_reset)
   END_RUNG
   // the same network as SCL:
   "Driver_Alerts_DB"(in_Robot_bLifeBit := "Robot".LifeBit,   // "Driver_Alerts"
                      in_Robot_bAlarmStop := "Robot".ALARM_STOP_KRC,
                      in_Robot_bUserSafe := "Robot".USER_SAF_KRC,
                      out_bAlarmReset => #Alarm_reset);
END_REGION

REGION Network 5
   RUNG wire#powerrail
      Move(in := "Robot_Programs", out1 => "Working_Programs")
   END_RUNG
   // the same network as SCL:
   "Working_Programs" := "Robot_Programs";
END_REGION

REGION Network 6
   RUNG wire#powerrail
      "Working_DB"(in_bStartButtonPushed :=, in_bEnableReturnTask := TRUE, in_bCountTriesReset := TRUE, in_usiCountTries := 1, in_iRequired := 1, in_bAlarm := #Alarms_out, in_bAlarmReset := #Alarm_reset, in_bInHome := "Robot".IN_HOME_KRC, in_bProgReq := "Robot".PGNO_REQ_KRC, in_bResume := false, in_bCancelTask := false, in_bModeDebug := false, in_pointer_array :=, in_Task := "WorkingTasks".Robot1, in_usiTaskStatus :=, in_bDebugNextStep :=, out_bStart =>, out_bStop =>, out_usiProgrammNumber =>, out_uiZoneFrom =>, out_uiZoneTo =>, out_uiRequired =>, out_A_bCantWork =>, out_usiCountTries =>, out_strJobStatus =>)
   END_RUNG
   // the same network as SCL:
   "Working_DB"(in_bEnableReturnTask := TRUE,   // "Driver_Working"
                in_bCountTriesReset := TRUE,
                in_usiCountTries := 1,
                in_iRequired := 1,
                in_bAlarm := #Alarms_out,
                in_bAlarmReset := #Alarm_reset,
                in_bInHome := "Robot".IN_HOME_KRC,
                in_bProgReq := "Robot".PGNO_REQ_KRC,
                in_bResume := false,
                in_bCancelTask := false,
                in_bModeDebug := false,
                in_Task := "WorkingTasks".Robot1);
END_REGION

REGION Network 8
   RUNG wire#powerrail
      "Matrix"()
   END_RUNG
   // the same network as SCL:
   "Matrix"();
END_REGION

REGION Network 9
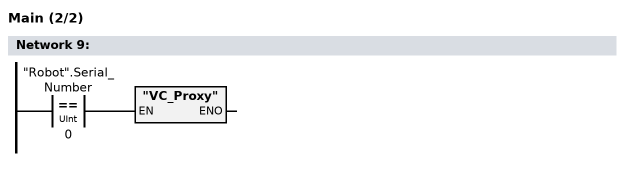
   RUNG wire#powerrail
      { S7_Templates := "SrcType := UInt" } EQ_Contact(in1 := "Robot".Serial_Number, in2 := 0)
      "VC_Proxy"()
   END_RUNG
   // the same network as SCL:
   IF "Robot".Serial_Number = 0 THEN "VC_Proxy"(); END_IF;
END_REGION
END_ORGANIZATION_BLOCK

ORGANIZATION_BLOCK "Cyclic interrupt"   // OB30, LAD, CyclicInterrupt
{ S7_Optimized_Access := 'TRUE' }
VERSION : 0.1
   VAR_INPUT
      Initial_Call : Bool;   // Initial call of this OB
      Event_Count : Int;   // Events discarded
   END_VAR
BEGIN
END_ORGANIZATION_BLOCK

ORGANIZATION_BLOCK "ProDiagOB"   // OB250, ProDiag_OB, ProgramCycle
TITLE = "Main Program Sweep (Cycle)"
{ S7_Optimized_Access := 'TRUE' }
VERSION : 0.1
   VAR_INPUT
      Initial_Call : Bool;   // Initial call of this OB
      Remanence : Bool;   // =True, if remanent data are available
   END_VAR
BEGIN

REGION Network 1
   CALL "Default_SupervisionFB", "Default_SupervisionDB";
END_REGION
END_ORGANIZATION_BLOCK

// folder: 1_Alerts

FUNCTION_BLOCK "Driver_Alerts"   // FB50, SCL
{ S7_Optimized_Access := 'TRUE' }
VERSION : 0.1
   VAR_INPUT
      in_bAlarmReset : Bool;   // Сброс Аварии
      in_bAlarmButton : Bool;   // Аварийная кнопка
      in_bPressureLoss : Bool;   // Низкое давление на входе
      in_bCantContinueTask : Bool;   // Не возможно продолжать работу
      in_Gripper_bTooLow : Bool;   // Захват. Ниже допустимой точки
      in_Gripper_bSheetLost : Bool;   // Захват. Лист потерян
      in_Gripper_bSheetTakeFail : Bool;   // Захват. Ошибка взятия листа
      in_Robot_bLifeBit : Bool;   // Робот. Бит жизни робота
      in_Robot_bAlarmStop : Bool;   // Робот. Аварийный останов
      in_Robot_bUserSafe : Bool;   // Робот. Защита пользователя
      in_Camera_bCantFind : Bool;   // Камера. Ошибка захвата изображения
      in_bDebugMode : Bool;   // DebugMode
   END_VAR
   VAR_OUTPUT
      out_Alarms : "Alarm";   // Аварии
      out_bAlarmReset : Bool;
   END_VAR
   VAR
      Static_Alarm : "Alarm";
      _bWarningReset : Bool;
      tLifeBitOn : TON_TIME;
      tLifeBitOff : TON_TIME;
      tWarningReset : TON_TIME;
      rtGripperTooDown : R_TRIG;
      rtGripperSheetLost : R_TRIG;
      rtGripperSheetTakeFail : R_TRIG;
      rtAlarm : R_TRIG;
   END_VAR
BEGIN
   ////////////////////////////Сброс Аварий и Предупреждениq///////////////////////////
   //Сброс Предупреждений
   #tWarningReset(IN := #Static_Alarm.bGenWarning AND NOT #_bWarningReset,
                      PT := T#500ms);
   IF #tWarningReset.Q THEN
       #_bWarningReset := TRUE;
   END_IF;
   IF #_bWarningReset THEN
       #Static_Alarm.W_bRobotSubmitDown := FALSE;
       #Static_Alarm.W_bRobotStop := FALSE;
       #Static_Alarm.W_bRobotUserSafe := FALSE;
       #Static_Alarm.W_bGripperTooDown := FALSE;
       #Static_Alarm.W_bGripperSheetLost := FALSE;
       #Static_Alarm.W_bGripperSheetTakeFail := FALSE;
       #Static_Alarm.W_bCameraCantFind := FALSE;
       #_bWarningReset := FALSE;
   END_IF;

   //Сброс Аварий
   IF #in_bAlarmReset THEN
       #Static_Alarm.A_bAlarmButtonPushed := FALSE;
       #Static_Alarm.A_bPressureLoss := FALSE;
       #Static_Alarm.A_bCantContinueTask := FALSE;
   END_IF;
   //////////////////////////////////////////////////////////////////////////////////// 

   ///////////////////////////////////////Аварии///////////////////////////////////////
   ///////////////////////////Требует нажатия "Сброс Аварии"///////////////////////////
   //Аварийная кнопка
   #Static_Alarm.A_bAlarmButtonPushed := NOT #in_bAlarmButton;

   //Низкое давление на входе в спарку
   #Static_Alarm.A_bPressureLoss := #in_bPressureLoss;

   //Робот не может завершить задание
   #rtAlarm(CLK := #in_bCantContinueTask);
   IF #rtAlarm.Q THEN
       #Static_Alarm.A_bCantContinueTask := TRUE;
   END_IF;

   //Наличие Аварии
   IF #Static_Alarm.A_bAlarmButtonPushed OR #Static_Alarm.A_bPressureLoss OR #Static_Alarm.A_bCantContinueTask THEN
       #Static_Alarm.bGenAlarm := TRUE;
   ELSE
       #Static_Alarm.bGenAlarm := FALSE;
   END_IF;
   ////////////////////////////////////////////////////////////////////////////////////

   /////////////////////////////////////Предупреждения/////////////////////////////////
   //////////////////////////НЕ Требует нажатия "Сброс Аварии"/////////////////////////
   //Аварийный останов от KUKA
   IF NOT #in_Robot_bAlarmStop THEN
       #Static_Alarm.W_bRobotStop := TRUE;
   END_IF;

   //Сработала защита пользователя
   IF NOT #in_Robot_bUserSafe THEN
       #Static_Alarm.W_bRobotUserSafe := TRUE;
   END_IF;

   //Submit остановлен
   #tLifeBitOn(IN := #in_Robot_bLifeBit,
                   PT := T#5s);
   #tLifeBitOff(IN := NOT #in_Robot_bLifeBit,
                    PT := T#5s);
   IF #tLifeBitOn.Q OR #tLifeBitOff.Q THEN
       #Static_Alarm.W_bRobotSubmitDown := TRUE;
   END_IF;

   //Защита от вдавливания
   #rtGripperTooDown(CLK := #in_Gripper_bTooLow);
   IF #rtGripperTooDown.Q THEN
       #Static_Alarm.W_bGripperTooDown := TRUE;
   END_IF;

   //Захват лист потерян во время движения
   #rtGripperSheetLost(CLK := #in_Gripper_bSheetLost);
   IF #rtGripperSheetLost.Q THEN
       #Static_Alarm.W_bGripperSheetLost := TRUE;
   END_IF;

   //Захват не смог взять #_A_Gripper_bSheetTakeFail
   #rtGripperSheetTakeFail(CLK := #in_Gripper_bSheetTakeFail);
   IF #rtGripperSheetTakeFail.Q THEN
       #Static_Alarm.W_bGripperSheetTakeFail := TRUE;
   END_IF;

   //Наличие Предупреждений
   IF #Static_Alarm.W_bRobotStop OR #Static_Alarm.W_bRobotUserSafe OR #Static_Alarm.W_bRobotSubmitDown OR
       #Static_Alarm.W_bGripperTooDown OR #Static_Alarm.W_bGripperSheetLost OR #Static_Alarm.W_bGripperSheetTakeFail THEN
       #Static_Alarm.bGenWarning := TRUE;
   ELSE
       #Static_Alarm.bGenWarning := FALSE;
   END_IF;
   ////////////////////////////////////////////////////////////////////////////////////

   ///////////////////////////////////Выходные данные//////////////////////////////////
   #Static_Alarm.bSTOP := #Static_Alarm.bGenWarning OR #Static_Alarm.bAlarmReset;
   ////////////////////////////////////////////////////////////////////////////////////

   ///////////////////////////////////Выходные данные//////////////////////////////////
   #out_Alarms := #Static_Alarm;
   #out_bAlarmReset := #tWarningReset.Q OR #in_bAlarmReset;
   ////////////////////////////////////////////////////////////////////////////////////
END_FUNCTION_BLOCK

// folder: 2_Robot

FUNCTION_BLOCK "Driver_RobotExternalStart"   // FB21, SCL
{ S7_Optimized_Access := 'TRUE' }
VERSION : 0.1
   VAR_INPUT
      in_bStart : Bool;
      in_bStop : Bool;
      in_Programm_iNubmer : Int;
      KRC_PLC_APPL_RUN : Int;
      KRC_PLC_PGNO_REQ : Bool;
      KRC_PLC_PRO_ACT : Bool;
      KRC_PLC_STOPMESS : Bool;
      KRC_PLC_PERI_RDY : Bool;
      KRC_PLC_ALARM_STOP : Bool;
      KRC_PLC_EXT_ACTIVE : Bool;
      KRC_PLC_USER_SAF : Bool;
      KRC_PLC_ON_PATH : Bool;
      KRC_PLC_IN_HOME : Bool;
      KRC_PLC_EXT_FIRST_START : Bool;
   END_VAR
   VAR_OUTPUT
      out_PGNO : Int;   // Номер программы
      PLC_KRC_PGNO_PARITY : Bool;
      PLC_KRC_PGNO_VALID : Bool;
      PLC_KRC_EXT_START : Bool;
      PLC_KRC_CONF_MESS : Bool;
      PLC_KRC_DRIVES_ON : Bool;
      PLC_KRC_DRIVES_OFF : Bool;
      PLC_KRC_MOVE_ENABLE : Bool;
   END_VAR
   VAR_IN_OUT
      in_Task : "TypeRobotTask";
   END_VAR
   VAR
      _iStatus : Int;
      _iStep_Start : Int;
      _iStep_DynamicBraking : Int;
      TStep_Start : Array[0..5] of TON_TIME;
      TStep_DynamicBraking : Array[0..5] of TON_TIME;
      i_Step_Start : Int;
      i_Step_DynamicBraking : Int;
   END_VAR
BEGIN
   /////////////////////////////////////////Инициализация/////////////////////////////////////////
   IF #_iStatus = 0 THEN
       #PLC_KRC_MOVE_ENABLE := TRUE;
       #PLC_KRC_DRIVES_OFF := TRUE;
       #PLC_KRC_CONF_MESS := FALSE;
       #PLC_KRC_DRIVES_ON := FALSE;
       #out_PGNO:=0;
   END_IF;
   //////////////////////////////////////////////////////////////////////////////////////////////

   ////////////////////////////////////////Выбор состояния///////////////////////////////////////
   //Состояние 1: Готов к заданию
   IF #KRC_PLC_USER_SAF AND #PLC_KRC_MOVE_ENABLE AND #KRC_PLC_ALARM_STOP AND
       #PLC_KRC_DRIVES_OFF AND NOT #PLC_KRC_DRIVES_ON AND #KRC_PLC_PERI_RDY AND
       NOT #PLC_KRC_CONF_MESS AND NOT #KRC_PLC_STOPMESS AND #KRC_PLC_PRO_ACT THEN
       #_iStatus := 1;

   //Состояние 2: Перезапуск после срабатывания Защиты пользователя
   ELSIF (#KRC_PLC_EXT_FIRST_START OR #in_Task.robot_alarm_reset) AND (NOT #KRC_PLC_USER_SAF OR NOT #KRC_PLC_PERI_RDY OR NOT #KRC_PLC_PRO_ACT) THEN
       #_iStatus := 2;
   END_IF;
   //////////////////////////////////////////////////////////////////////////////////////////////

   ////////////////////////////////////////Флаг перезапуска после ошибки///////////////////////////////////////
   //Сброс флага
   #in_Task.robot_alarm_reset := FALSE;

   /////////////////////////////////////////Логика работы////////////////////////////////////////
   //Состояние 1: Готов к заданию
   IF #_iStatus = 1 THEN
       //ШАГ 1: Отправляем бит "Старт с внешней автоматики"
       IF #_iStep_Start = 0 AND #in_bStart AND #KRC_PLC_PGNO_REQ THEN
           #_iStep_Start := 1;

       END_IF;

       //ШАГ 2: Подтверждаем валидность программы
       IF #TStep_Start[1].ET > T#100ms THEN
           #_iStep_Start := 2;
       END_IF;

       //ШАГ 0: При завершении программы снимаем Валидность и Паритет программы
       IF #TStep_Start[2].ET > T#100ms AND (NOT #KRC_PLC_PGNO_REQ OR #in_Programm_iNubmer<>#out_PGNO) THEN
           #_iStep_Start := 0;
       END_IF;

       CASE #_iStep_Start OF
           0: //ШАГ 0: Выставляем параметры по дефолту
               #PLC_KRC_EXT_START := FALSE;
               #PLC_KRC_PGNO_VALID := FALSE;
               #PLC_KRC_PGNO_PARITY := FALSE;

           1: //ШАГ 1: Отправляем бит "Старт с внешней автоматики"
               #out_PGNO := #in_Programm_iNubmer; //Номер программы

           2: //ШАГ 2: Подтверждаем валидность программы
               #PLC_KRC_PGNO_VALID := "Robot"."PGNO_REFL_KRC"="To_KUKA_PGNO_KRC" AND "To_KUKA_PGNO_KRC"<>0;
               //#PLC_KRC_PGNO_VALID := TRUE;

       END_CASE;
   ELSE
       #_iStep_Start := 0;
   END_IF;

   //Состояние 2: Перезапуск после срабатывания Защиты пользователя
   IF #_iStatus = 2 THEN
       //ШАГ 0: Предподготовка 
       IF #TStep_DynamicBraking[0].Q OR #TStep_DynamicBraking[1].Q OR 
           #TStep_DynamicBraking[2].Q OR #TStep_DynamicBraking[3].Q THEN
           #_iStep_DynamicBraking := 0;
       END_IF;

       //ШАГ 1: Включаем привода
       IF #TStep_DynamicBraking[0].ET > T#200ms AND #KRC_PLC_USER_SAF AND #KRC_PLC_ALARM_STOP THEN
           #_iStep_DynamicBraking := 1;
       END_IF;

       //ШАГ 2: Снимаем стоповый бит
       IF #TStep_DynamicBraking[1].ET > T#200ms AND #KRC_PLC_PERI_RDY AND #KRC_PLC_USER_SAF AND #KRC_PLC_ALARM_STOP THEN
           #_iStep_DynamicBraking := 2;
       END_IF;

       //ШАГ 3: Запускаем программу
       IF #TStep_DynamicBraking[2].ET > T#200ms AND NOT #KRC_PLC_STOPMESS AND #KRC_PLC_USER_SAF AND #KRC_PLC_ALARM_STOP AND NOT #in_bStop THEN
           #_iStep_DynamicBraking := 3;
       END_IF;

       CASE #_iStep_DynamicBraking OF
           0:  //ШАГ 0: Предподготовка
               #PLC_KRC_DRIVES_ON := FALSE;
               #PLC_KRC_CONF_MESS := FALSE;
               #PLC_KRC_EXT_START := FALSE;

           1: //ШАГ 1: Включаем привода
               #PLC_KRC_DRIVES_ON := TRUE;
               #PLC_KRC_CONF_MESS := TRUE;

           2: //ШАГ 2: Снимаем стоповый бит
               #PLC_KRC_DRIVES_ON := FALSE;
               #PLC_KRC_CONF_MESS := FALSE;

           3: //ШАГ 3: Запускаем программу
               #PLC_KRC_EXT_START := TRUE;
       END_CASE;
   ELSE
       #_iStep_DynamicBraking := 0;
       IF #_iStatus <> 3 OR #_iStatus <> 4 THEN
           #PLC_KRC_EXT_START := FALSE;
       END_IF;
   END_IF;
   //////////////////////////////////////////////////////////////////////////////////////////////

   ////////////////////////////////////////////Таймеры///////////////////////////////////////////
   //Запуск 
   #TStep_Start[#_iStep_Start](IN := TRUE,
                               PT := T#10m);
   #TStep_DynamicBraking[#_iStep_DynamicBraking](IN := TRUE,
                                                 PT := T#10s);
   //Останов
   FOR #i_Step_Start := 0 TO 5 DO
       IF #_iStep_Start <> #i_Step_Start THEN
           #TStep_Start[#i_Step_Start](IN := FALSE,
                                       PT := T#10s);
       END_IF;
   END_FOR;
   FOR #i_Step_DynamicBraking := 0 TO 5 DO
       IF #_iStep_DynamicBraking <> #i_Step_DynamicBraking THEN
           #TStep_DynamicBraking[#i_Step_DynamicBraking](IN := FALSE,
                                                         PT := T#10s);
       END_IF;
   END_FOR;
   //////////////////////////////////////////////////////////////////////////////////////////////
END_FUNCTION_BLOCK

FUNCTION_BLOCK "Driver_RobotPause"   // FB22, SCL
{ S7_Optimized_Access := 'TRUE' }
VERSION : 0.1
   VAR_INPUT
      in_bPauseButton : Bool;   // Кнопка пауза Физическая
      in_bHMIPause : Bool;   // Кнопка пауза HMI
   END_VAR
   VAR_OUTPUT
      out_bPause : Bool;   // Пауза
      out_bPauseStatus : Bool;   // Пауза
   END_VAR
   VAR
      _bPause : Bool;   // Пауза
      rtPauseOn : R_TRIG;   // Тригер паузы
   END_VAR
BEGIN
   #rtPauseOn(CLK := #in_bPauseButton);
   IF #rtPauseOn.Q AND #_bPause THEN
       #_bPause := FALSE;
   ELSIF #rtPauseOn.Q AND NOT #_bPause THEN
       #_bPause := TRUE;
   END_IF;
   #out_bPause := #_bPause;
END_FUNCTION_BLOCK

FUNCTION_BLOCK "!Robot"   // FB200, SCL
{ S7_Optimized_Access := 'TRUE' }
VERSION : 0.1
BEGIN
   /////////////////////////////////////////Робот - Пауза////////////////////////////////////////
   "RobotPause_DB"(in_bPauseButton := FALSE,
                   in_bHMIPause:=FALSE);
   //////////////////////////////////////////////////////////////////////////////////////////////

   ///////////////////////////////////Режим внешней Автоматики///////////////////////////////////
   "RobotExternalStart"(in_bStart := "Working_DB".out_bStart,
                        in_bStop := "Alerts_DB".out_Alarms.bGenAlarm,
                        in_Programm_iNubmer := "Working_DB".out_usiProgrammNumber,
                        KRC_PLC_APPL_RUN:=0,
                        KRC_PLC_ON_PATH:=false,
                        in_Task := "RobotTasks".Robot1,
                        KRC_PLC_PGNO_REQ := "Robot"."PGNO_REQ_KRC",
                        KRC_PLC_PRO_ACT := "Robot"."PRO_ACT_KRC",
                        KRC_PLC_STOPMESS := "Robot"."STOPMESS_KRC",
                        KRC_PLC_PERI_RDY := "Robot"."PERI_RDY_KRC",
                        KRC_PLC_ALARM_STOP := "Robot"."ALARM_STOP_KRC",
                        KRC_PLC_EXT_ACTIVE := "Robot"."EXT_ACTIVE",
                        KRC_PLC_USER_SAF := "Robot"."USER_SAF_KRC",
                        KRC_PLC_IN_HOME := "Robot"."IN_HOME_KRC",
                        KRC_PLC_EXT_FIRST_START := "Robot"."EXT_FIRST_START",
                        out_PGNO => "KUKA_Data".PGNO_KRC,
                        PLC_KRC_PGNO_PARITY => "To_KUKA_PGNO_PARITY",
                        PLC_KRC_PGNO_VALID => "To_KUKA_PGNO_VALID_KRC",
                        PLC_KRC_EXT_START => "To_KUKA_EXT_START_KRC",
                        PLC_KRC_CONF_MESS => "To_KUKA_CONF_MESS",
                        PLC_KRC_DRIVES_ON => "To_KUKA_DRIVERS_ON",
                        PLC_KRC_DRIVES_OFF => "To_KUKA_DRIVERS_OFF",
                        PLC_KRC_MOVE_ENABLE => "To_KUKA_MOVE_ENABLE_KRC");

   //////////////////////////////////////////////////////////////////////////////////////////////

   //Обмен данными PLC, KUKA  ------- Перенести в IO
   "KUKA_IO_DB"();
END_FUNCTION_BLOCK

FUNCTION_BLOCK "KUKA_IO"   // FB204, SCL
{ S7_Optimized_Access := 'TRUE' }
VERSION : 0.1
BEGIN
   ///////////////////////////KUKA 1//////////////////////////////
   //DATA To PLC From KUKA
   //"KUKA_Data".PGNO_REFL_KRC := ROR(IN := "From_KUKA_PGNO_REFL_KRC", N := 8);
   //"Task".robot_A1 := ROR(IN := "From_KUKA_A1_Angle_plus_180", N := 8) - 180;
   //"Task".robot_Z := ROR(IN := "From_KUKA_Pos_Z", N := 8);


   //DATA To KUKA From PLC
   IF "To_KUKA_PLC_STOP" THEN
       "KUKA_Data".PGNO_KRC := 0;
   END_IF;

   "To_KUKA_PGNO_KRC" := ROR(IN := "KUKA_Data".PGNO_KRC, N := 8);

   //"To_KUKA_PLC_STOP" := FALSE;
   //"To_KUKA_PAUSE_STOP" := "RobotPause_DB".out_bPause;
   ///////////////////////////////////////////////////////////////
END_FUNCTION_BLOCK

FUNCTION "CrossConnection" : Void   // FC1, SCL
{ S7_Optimized_Access := 'TRUE' }
VERSION : 0.1
   VAR_TEMP
      button_Pause_pressed : Bool;
      button_Start_pressed : Bool;
      button_Reset_withheld : Bool;
      button_Reset_reset : Bool;
      button_Start_withheld : Bool;
      button_Start_reset : Bool;
      Start_elapsed_time : Time;
      Reset_elapsed_time : Time;
      Cnt : UInt;
   END_VAR
BEGIN
   "To_KUKA_IsGripperMainHome" := "InGripperMainHome1" AND "InGripperMainHome2";
   "To_KUKA_IsGripperFeederHome" := "InGripperFeederHome" ;
   "To_KUKA_GripperRetracted" := "InGripperRetracted";
   "To_KUKA_Gercon" := NOT "InGripperGerconNC";
   "To_KUKA_Collision" := FALSE;
   "To_KUKA_Vacuum_Ok" := NOT "InGripperVacuumNC";
   "To_KUKA_WithoutMachine" := "RobotTasks".Robot1."w/o_machine_mode";
   "OutVacuumON" := "Robot"."SetVacuumON";
   "OutPressureOFF" := "Robot"."SetPressureOFF";
   "OutGripperMainRetract" := "Robot"."SetRetract";
   "OutFlow2Part" := "Robot"."Flow2PartON";
   "OutFlipClose" := "Robot"."SetFlipClose";
   "OutFlipVacuumOn" := "Robot"."FlipVacuumOn";

   "PLC_WorkpieceAtStopper" := "WorkpieceAtStopper";
   "PLC_InfeedAreaFree" := "InfeedAreaFree";
   "PLC_OutfeedAreaFree" := "OutfeedAreaFree";
   "PLC_OpenClamps" := "OpenClamps";
   "PLC_ResetMcc" := "ResetMcc";
   "InfeedPositionFree" := "PLC_InfeedPositionFree";
   "WorkpieceClamped" := "PLC_WorkpieceClamped";
   "WorkpieceRdyToTurn" := "PLC_WorkpieceRdyToTurn";
   "WorkpiecePickupPos1" := "PLC_WorkpiecePickupPos1";
   "WorkpiecePickupPos2" := "PLC_WorkpiecePickupPos2";
   "AutoFeedingModeActive" := "PLC_AutoFeedingModeActive";
   "StopperWorkpos" := "PLC_StopperWorkpos";


   //"To_KUKA_Part_length_X" := ROR(IN := "RobotTasks".Robot1.part_length_X, N := 8);
   //"To_KUKA_Part_length_Y" := ROR(IN := "RobotTasks".Robot1.part_length_Y, N := 8);
   //"To_KUKA_Part_thickness_Z" := ROR(IN := "RobotTasks".Robot1.part_thickness_Z, N := 8);
   //"To_KUKA_QRcode_X" := ROR(IN := "RobotTasks".Robot1.label_pos_X, N := 8);
   //"To_KUKA_QRcode_Y" := ROR(IN := "RobotTasks".Robot1.label_pos_Y, N := 8);
   //"To_KUKA_QRcode_Angle" := ROR(IN := "RobotTasks".Robot1.label_pos_A, N := 8);
   "To_KUKA_Rangefinder" := ROR(IN := "InGripperRangefinder", N := 8);
   "To_KUKA_Part_Length_X0" := ROR(IN := "RobotTasks".Robot1.part_length_X0, N := 8);
   "To_KUKA_Part_Length_Y0" := ROR(IN := "RobotTasks".Robot1.part_length_Y0, N := 8);
   "To_KUKA_Part_length_X" := ROR(IN := "RobotTasks".Robot1.part_length_X, N := 8);
   "To_KUKA_Part_length_Y" := ROR(IN := "RobotTasks".Robot1.part_length_Y, N := 8);
   "To_KUKA_Part_thickness_Z" := ROR(IN := "RobotTasks".Robot1.part_thickness_Z, N := 8);
   "To_KUKA_Part_Slot" := ROR(IN := USINT_TO_UINT("RobotTasks".Robot1.part_slot), N := 8);
   "To_KUKA_Free_Slot" := ROR(IN := USINT_TO_UINT("RobotTasks".Robot1.free_slot), N := 8);

   "To_KUKA_Gripper_Sign_X" := "RobotTasks".Robot1.gripper_sign_X;
   "To_KUKA_Gripper_Sign_Y" := "RobotTasks".Robot1.gripper_sign_Y;


   "To_KUKA_Gripper_Within_part":="RobotTasks".Robot1.gripper_within_part;

   "To_KUKA_PAUSE_STOP" := "RobotTasks".Robot1.robot_pause;




   IF "Robot"."Pallet_Scanned" THEN
       IF NOT "To_KUKA_AckPalletScanned" THEN
           "RobotTasks".Robot1."pallet_scanned" := TRUE;
           "To_KUKA_AckPalletScanned" := TRUE;
       END_IF;
   ELSE
       "To_KUKA_AckPalletScanned" := FALSE;
   END_IF;


   "Set_OUT"(In_val := "RobotTasks".Robot1.part_pos_X,
             Out_val := "To_KUKA_Part_X");
   "Set_OUT"(In_val := "RobotTasks".Robot1."part_pos_Y",
             Out_val := "To_KUKA_Part_Y");
   "Set_OUT"(In_val := "RobotTasks".Robot1."part_pos_Z",
             Out_val := "To_KUKA_Part_Z");
   "Set_OUT"(In_val := "RobotTasks".Robot1."part_angle_A",
             Out_val := "To_KUKA_Part_A");

   "Set_OUT"(In_val := "RobotTasks".Robot1.slot_pos_X,
             Out_val := "To_KUKA_Slot_X");
   "Set_OUT"(In_val := "RobotTasks".Robot1."slot_pos_Y",
             Out_val := "To_KUKA_Slot_Y");
   "Set_OUT"(In_val := "RobotTasks".Robot1."slot_pos_Z",
             Out_val := "To_KUKA_Slot_Z");
   "Set_OUT"(In_val := "RobotTasks".Robot1."slot_angle_A",
             Out_val := "To_KUKA_Slot_A");

   "Set_OUT"(In_val := "RobotTasks".Robot1.out_pos_X,
             Out_val := "To_KUKA_Out_X");
   "Set_OUT"(In_val := "RobotTasks".Robot1."out_pos_Y",
             Out_val := "To_KUKA_Out_Y");
   "Set_OUT"(In_val := "RobotTasks".Robot1."out_pos_Z",
             Out_val := "To_KUKA_Out_Z");
   "Set_OUT"(In_val := "RobotTasks".Robot1."out_pos_A",
             Out_val := "To_KUKA_Out_A");

   "RobotTasks".Robot1.robot_serial := "Robot"."Serial_Number";





   "RobotTasks".Robot1.robot_in_home:="Robot"."IN_HOME_KRC";

   //Статус машины
   IF "RobotTasks".Robot1."w/o_machine_mode" THEN
       //machine shunt
       IF "RobotTasks".Robot1.robot_program = 7 THEN
           "RobotTasks".Robot1.machine_status := 'ready2unload';
       ELSE
           "RobotTasks".Robot1.machine_status := 'ready2load';
       END_IF;
   ELSE
       IF "PLC_InfeedPositionFree" AND "PLC_AutoFeedingModeActive" AND "PLC_StopperWorkpos" AND NOT "PLC_WorkpieceClamped" THEN
           "RobotTasks".Robot1.machine_status:='ready2load';
       ELSIF "PLC_WorkpiecePickupPos2" AND "PLC_AutoFeedingModeActive" AND "PLC_WorkpieceClamped" THEN
           "RobotTasks".Robot1.machine_status := 'ready2unload';
       ELSIF NOT "PLC_AutoFeedingModeActive" THEN
           "RobotTasks".Robot1.machine_status := 'manual_mode';
       ELSIF FALSE THEN
           "RobotTasks".Robot1.machine_status := 'busy';
       ELSIF "RobotTasks".Robot1.machine_status = '' THEN
           "RobotTasks".Robot1.machine_status := 'unknown';
       ELSE
           "RobotTasks".Robot1.machine_status := 'unknown';
       END_IF;
   END_IF;

   //Статус робота
   IF "Robot"."PRO_MOVE_KRC" THEN
       "RobotTasks".Robot1.robot_status := 'busy';
   ELSIF NOT "Robot"."EXT_ACTIVE" THEN
       "RobotTasks".Robot1.robot_status := 'manual_mode';
   ELSIF "Robot"."EXT_ACTIVE" AND (NOT "Robot"."PRO_MOVE_KRC") AND "Robot"."IN_HOME_KRC" THEN
       "RobotTasks".Robot1.robot_status := 'home';
   ELSIF "Robot".AXIS_ACT_A1=82.5 OR
       ("Robot".AXIS_ACT_A1>50.0 AND  "Robot".AXIS_ACT_A1<120.0 AND "RobotTasks".Robot1.robot_trajectory = 'PartHeightMeasuring')  OR
       ("Robot".AXIS_ACT_A1>78.0 AND  "Robot".AXIS_ACT_A1<93.0) THEN
       //machine shunt
       IF "RobotTasks".Robot1."w/o_machine_mode" THEN
           IF "RobotTasks".Robot1.robot_trajectory = 'UnloadMachine' THEN
               "RobotTasks".Robot1.part_status := 'gripper';
               "RobotTasks".Robot1.robot_status := 'pallet_out';
           ELSIF "RobotTasks".Robot1.robot_trajectory = 'LoadMachine' THEN
               "RobotTasks".Robot1.robot_status := 'at_machine';
               "RobotTasks".Robot1.part_status := 'in_machine';
               //ELSIF "RobotTasks".Robot1.robot_program = 3 THEN
               //    "RobotTasks".Robot1.robot_status := 'at_machine';
               //    "RobotTasks".Robot1.part_status := 'gripper';
           ELSE
               "RobotTasks".Robot1.robot_status := 'pallet_in';
           END_IF;
       ELSE
           "RobotTasks".Robot1.robot_status := 'pallet_in';
       END_IF;
   ELSIF  "Robot".AXIS_ACT_A1>-33.5 AND "Robot".AXIS_ACT_A1<10.0 THEN
       "RobotTasks".Robot1.robot_status := 'flip_table';
       //machine shunt
       IF "RobotTasks".Robot1."w/o_machine_mode" THEN
           IF "RobotTasks".Robot1.robot_trajectory = 'UnloadMachine' THEN
               "RobotTasks".Robot1.part_status := 'gripper';
               "RobotTasks".Robot1.robot_status := 'pallet_out';
           ELSIF "RobotTasks".Robot1.robot_trajectory = 'LoadMachine' THEN
               "RobotTasks".Robot1.robot_status := 'at_machine';
           END_IF;
       END_IF;
   ELSIF "Robot".AXIS_ACT_A1=35 THEN
       "RobotTasks".Robot1.robot_status := 'part_slot';
   ELSIF "Robot".AXIS_ACT_A1=-33.5 OR ("Robot".AXIS_ACT_A1>-60.0 AND "Robot".AXIS_ACT_A1<-50.0) THEN
       "RobotTasks".Robot1.robot_status := 'pallet_out';
   ELSIF "Robot".AXIS_ACT_A1>-108.0 AND "Robot".AXIS_ACT_A1<-105.0  THEN
       "RobotTasks".Robot1.robot_status := 'at_machine';
   ELSIF "RobotTasks".Robot1.robot_status='' THEN
       "RobotTasks".Robot1.robot_status := 'unknown';
   ELSIF "RobotTasks".Robot1.operation_type='go_home' THEN
       "RobotTasks".Robot1.robot_status := 'go_home';
   ELSE
       "RobotTasks".Robot1.robot_status := 'unknown';
   END_IF;

   //Сброс флага новой детали (чтобы не загружалась программа), если на станке работает оператор
   "RobotTasks".Robot1.not_sended2BHX := "RobotTasks".Robot1.not_sended2BHX AND "PLC_AutoFeedingModeActive";
   IF "RobotTasks".Robot1.not_sended2BHX AND "PLC_AutoFeedingModeActive" AND "RobotTasks".Robot1.program_fullpath<>'' THEN
       "RobotTasks".Robot1.not_sended2Arduino := TRUE;
       "RobotTasks".Robot1.not_sended2BHX := FALSE;
   END_IF;



   IF "RobotTasks".Robot1.robot_program>"Robot_Programs".Count THEN
       "RobotTasks".Robot1.robot_program := 0;
   END_IF;

   IF "RobotTasks".Robot1.reset_job THEN
       //IF "Robot"."IN_HOME_KRC" THEN
           "ResetJob"(in_Task:= "RobotTasks".Robot1);
       //END_IF;
   END_IF;

   //Кнопки
   "Pause_R_TRIG_DB"(CLK := "button_Pause",
                     Q => #button_Pause_pressed);

   IF #button_Pause_pressed THEN
       "RobotTasks".Robot1.robot_pause := NOT "RobotTasks".Robot1.robot_pause;
   END_IF;

   "Pallet_start_timer".TONR(IN:="button_Start",
                             PT:=T#3s,
                             R:="Timers".button_Start_R,
                             ET=>#Start_elapsed_time);

   "Start_R_TRIG_DB"(CLK:="Pallet_start_timer".Q,
                     Q=>#button_Start_withheld);

   IF "button_Start" THEN
       "Timers".button_Start_R := FALSE;
   END_IF;

   IF NOT "button_Start" THEN
       IF #Start_elapsed_time > T#0s AND #Start_elapsed_time < "Pallet_start_timer".PT THEN
           IF "RobotTasks".Robot1.robot_pause THEN
               "RobotTasks".Robot1.robot_pause := FALSE;
           ELSE
               "RobotTasks".Robot1.start_job := TRUE;
           END_IF;
       END_IF;
       "Timers".button_Start_R := TRUE;
   END_IF;

   IF #button_Start_withheld THEN
       //"RobotTasks".Robot1.reset_job := TRUE;
       "RobotTasks".Robot1.start_job := TRUE;
       "RobotTasks".Robot1.robot_pause := FALSE;
       //"RobotTasks".Robot1.new_pallet := TRUE;
       "Matrix_output".scan_lay_number := 2;
    END_IF;

   "Go_home_timer".TONR(IN := "button_Reset",
                        PT := T#5s,
                        R := "Timers".button_Reset_R,
                        ET => #Reset_elapsed_time);

   "Reset_R_TRIG_DB"(CLK:="Go_home_timer".Q,
                     Q=>#button_Reset_withheld);

   IF "button_Reset" THEN
       "Timers".button_Reset_R := FALSE;
   ELSE
       IF "To_KUKA_PLC_STOP" THEN
           "To_KUKA_PLC_STOP" := FALSE;
       END_IF;
       IF #Reset_elapsed_time > T#0s AND #Reset_elapsed_time < "Go_home_timer".PT THEN
           "RobotTasks".Robot1.robot_alarm_reset := TRUE;
       END_IF;
       "Timers".button_Reset_R := TRUE;
   END_IF;

   //IF "button_Reset" AND ("RobotTasks".Robot1.operation_type = 'go_home' OR "RobotTasks".Robot1.operation_type = '') THEN //"Robot"."PRO_ACT_KRC" AND "Robot"."EXT_ACTIVE" AND 
   //    //IF NOT "button_Reset" AND "RobotTasks".Robot1.task_status <> 'done' AND "RobotTasks".Robot1.operation_type <> 'finish' THEN
   //    //    ;
   //    //ELSE
   //        "To_KUKA_PLC_STOP" := FALSE;
   //    //END_IF;
   //END_IF;

   IF (#button_Reset_withheld AND "Robot"."PRO_ACT_KRC" AND "Robot"."EXT_ACTIVE") THEN
       "RobotTasks".Robot1.reset_job := TRUE;
       //"ResetJob"(in_Task:="RobotTasks".Robot1);
       IF NOT "Robot"."IN_HOME_KRC" THEN
           "To_KUKA_PLC_STOP" := TRUE;
           "RobotTasks".Robot1.new_pallet := TRUE;
           "RobotTasks".Robot1.robot_pause := FALSE;
       END_IF;
   END_IF;

   IF NOT "Robot"."EXT_ACTIVE" THEN
       "RobotTasks".Robot1.reset_job := FALSE;
       "RobotTasks".Robot1.start_job := FALSE;
   END_IF;

   //IF "button_Start" AND "RobotTasks".Robot1.task_status = 'in_process' AND ("RobotTasks".Robot1.operation_type = 'go_home' OR "RobotTasks".Robot1.operation_type = 'scanning') AND "Robot"."IN_HOME_KRC" THEN
   //    ;//"RobotTasks".Robot1.task_status := 'done';
   //END_IF;
   //

   Strg_TO_Chars(Strg := "RobotTasks".Robot1.task_status,
                 pChars := 0,
                 Cnt => #Cnt,
                 Chars := "task_status".str);

   Strg_TO_Chars(Strg := "RobotTasks".Robot1.part_status,
                 pChars := 0,
                 Cnt => #Cnt,
                 Chars := "part_status".str);
END_FUNCTION

FUNCTION "Set_OUT" : Void   // FC7, SCL
{ S7_Optimized_Access := 'TRUE' }
VERSION : 0.1
   VAR_INPUT
      In_val : Real;
   END_VAR
   VAR_IN_OUT
      Out_val : UInt;
   END_VAR
   VAR_TEMP
      Temp_val : UInt;
   END_VAR
BEGIN
   IF #In_val < 0 THEN
       #Temp_val := 65520 + #In_val*10;
   ELSE
       #Temp_val := #In_val*10;
   END_IF;

   #Out_val := ROR(IN := #Temp_val, N := 8);
END_FUNCTION

FUNCTION "Get_IN" : Void   // FC8, SCL
{ S7_Optimized_Access := 'TRUE' }
VERSION : 0.1
   VAR_INPUT
      In_val : UInt;
   END_VAR
   VAR_IN_OUT
      Out_val : Real;
   END_VAR
   VAR_TEMP
      Tmp_val : Real;
   END_VAR
BEGIN
   #Tmp_val:=ROR(IN := #In_val, N := 8)/10.0;
   IF #Tmp_val > 3276 THEN
       #Out_val := #Tmp_val-6552;
   ELSE
       #Out_val := #Tmp_val;
   END_IF;
END_FUNCTION

FUNCTION "Get_Robot_Program" : Void   // FC9, SCL
{ S7_Optimized_Access := 'TRUE' }
VERSION : 0.1
   VAR_INPUT
      in_Task : "TypeRobotTask";
   END_VAR
   VAR_OUTPUT
      Program_number : UInt;
   END_VAR
   VAR_TEMP
      i : UInt;
      j : UInt;
      operation_type_ok : Bool;
      machine_status_ok : Bool;
      robot_status_ok : Bool;
      part_status_ok : Bool;
      first_program_ok : Bool;
      previous_trajectory_ok : Bool;
      program_ok : Bool;
      lay_ok : Bool;
      operation_side_ok : Bool;
      part_side_ok : Bool;
      part_destination_ok : Bool;
      entryPoint_active : Bool;
   END_VAR
BEGIN
   #Program_number := 0;
   FOR #i := 1 TO "Robot_Programs".Count DO
       FOR #j := 1 TO 12 DO
           IF #Program_number=0 THEN
               #machine_status_ok := ("Robot_Programs".List[#i].Entry_Points[#j].machine_status = #in_Task.machine_status)
                   OR ("Robot_Programs".List[#i].Entry_Points[#j].machine_status = '');
                   #robot_status_ok := ("Robot_Programs".List[#i].Entry_Points[#j].robot_status = #in_Task.robot_status)
                   OR ("Robot_Programs".List[#i].Entry_Points[#j].robot_status = '');
                   #part_status_ok := ("Robot_Programs".List[#i].Entry_Points[#j].part_status = #in_Task.part_status)
                   OR ("Robot_Programs".List[#i].Entry_Points[#j].part_status = '');
                   #previous_trajectory_ok := "Robot_Programs".List[#i].Entry_Points[#j].previous_trajectory = #in_Task.robot_trajectory;
               #first_program_ok := "Robot_Programs".List[#i].Entry_Points[#j].previous_trajectory = '';
               #operation_type_ok := "Robot_Programs".List[#i].Entry_Points[#j].operation_type = #in_Task.operation_type;
               #program_ok := #previous_trajectory_ok OR #first_program_ok OR #i = #in_Task.robot_program;
               #lay_ok := ("Robot_Programs".List[#i].Entry_Points[#j].lay_number = #in_Task.lay_number)
                   OR ("Robot_Programs".List[#i].Entry_Points[#j].lay_number = -1);
               #operation_side_ok := ("Robot_Programs".List[#i].Entry_Points[#j].operation_side = #in_Task.operation_side)
                   OR ("Robot_Programs".List[#i].Entry_Points[#j].operation_side = '');
               #part_side_ok := ("Robot_Programs".List[#i].Entry_Points[#j].part_side = #in_Task.part_side)
                   OR ("Robot_Programs".List[#i].Entry_Points[#j].part_side = '');
               #part_destination_ok := ("Robot_Programs".List[#i].Entry_Points[#j].part_destination = #in_Task.part_destination)
                   OR ("Robot_Programs".List[#i].Entry_Points[#j].part_destination = '');
               #entryPoint_active := "Robot_Programs".List[#i].Entry_Points[#j].active;
               IF #operation_type_ok AND #machine_status_ok AND #robot_status_ok AND #part_status_ok AND #part_destination_ok
                   AND #program_ok AND #lay_ok AND #operation_side_ok AND #part_side_ok AND #entryPoint_active THEN
                   #Program_number := #i;
               END_IF;
               IF #i="Get_Robot_Program_DB".i AND #j="Get_Robot_Program_DB".j THEN
                   "Get_Robot_Program_DB".operation_type_ok:=#operation_type_ok;
                   "Get_Robot_Program_DB".machine_status_ok:=#machine_status_ok;
                   "Get_Robot_Program_DB".robot_status_ok:=#robot_status_ok;
                   "Get_Robot_Program_DB".part_status_ok:=#part_status_ok;
                   "Get_Robot_Program_DB".first_program_ok:=#first_program_ok;
                   "Get_Robot_Program_DB".previous_trajectory_ok:= #previous_trajectory_ok;
                   "Get_Robot_Program_DB".program_ok:=#program_ok;
                   "Get_Robot_Program_DB".lay_ok:=#lay_ok;
                   "Get_Robot_Program_DB".operation_side_ok:=#operation_side_ok;
                   "Get_Robot_Program_DB".part_side_ok:=#part_side_ok;
                   "Get_Robot_Program_DB".part_destination_ok:=#part_destination_ok;
                   "Get_Robot_Program_DB".entryPoint_active:=#entryPoint_active;
               END_IF;
           END_IF;
       END_FOR;
   END_FOR;
END_FUNCTION

// folder: 3_Gripper

FUNCTION_BLOCK "Driver_Gripper"   // FB31, SCL
{ S7_Optimized_Access := 'TRUE' }
VERSION : 0.1
   VAR_INPUT
      in_usiCountTries : USInt;
      in_bRobotExtControl : Bool;
      in_DebugMode : Bool;
   END_VAR
   VAR_OUTPUT
      out_A_bSheetLost : Bool;   // Авария. Лист потерян при перемещении
      out_A_bSheetTakeFail : Bool;   // Авария. Не возможно взять лист
   END_VAR
   VAR
      _usiVacuum : USInt;   // Кол-во рабочих датчиков Вакууума
      _iWorkStatus : USInt;   // Статус работы
      _bSheetPressent : Bool;
      _bLoadingOK : Bool;
      _bUnLoadingOK : Bool;
      _Vacuum_bOn : Bool;   // Вакуум. Группа 1. Включить
      _bWaitingUnloading : Bool;   // Ожидает разгрузку
      _A_bSheetLost : Bool;
      _A_bSheetTakeFail : Bool;
      _usiCountTries : USInt;   // Количество попыток взятия листа
      _usiStepReady : USInt;
      _usiStepLoading : USInt;   // Шаги загрузки
      tBlowAfterLoad : TOF_TIME;
      tStepLoading : Array[0..15] of TON_TIME;
      i_tStepLoading : USInt;
      _usiStepUnLoading : USInt;   // Шаги разгрузки
      tStepUnLoading : Array[0..15] of TON_TIME;
      i_tStepUnLoading : USInt;
      tbWaitingUnloading : TON_TIME;
      tAlarmSheetLost : TOF_TIME;
      rtCountTries : R_TRIG;
      rtVacuumOn : R_TRIG;
   END_VAR
   VAR CONSTANT
      Status_Ready : USInt := 1;   // Статус. Ожидание команды
      Status_Loading : USInt := 2;   // Статус. Загрузка
      Status_UnLoading : USInt := 3;   // Статус. Разгрузка
      Step_Ready : USInt := 0;   // Шаг. Готовность
      Step_PreStart : USInt := 1;   // Шаг. Подготовка
      Step_VacuumOn : USInt := 3;   // Шаг. Включаем Вакуум
      Step_LoadingOk : USInt := 6;   // Шаг. Загрузка ОК
      Step_UnLoadingOk : USInt := 8;   // Шаг. Разгрузка ОК
      cSheetNonCovered : USInt := 0;
      cSheetCovered : USInt := 1;
      cSheetSubstrate : USInt := 2;
      cSheetInvalidCover : USInt := 3;
      cMaxCountTries : USInt := 2;
      cDelayUnloadVacuumOn : Time := T#200MS;
      cDelayUnloadVacuumOff : Time := T#200MS;
   END_VAR
BEGIN

   #_bSheetPressent := NOT "InGripperGerconNC";
   //////////////////////////////////////Защиты и Блокировки/////////////////////////////////////
   //Ошибка взятия листа
   #_A_bSheetTakeFail := #_usiCountTries >= #cMaxCountTries;
   #_A_bSheetLost := #_bWaitingUnloading AND NOT #_bSheetPressent;

   //Отключение вакуума после аварии
   IF #_A_bSheetTakeFail OR #_A_bSheetLost THEN
       #_Vacuum_bOn := FALSE;
   END_IF;
   //////////////////////////////////////////////////////////////////////////////////////////////

   ////////////////////////////////////////Выбор состояния///////////////////////////////////////
   //IF NOT #in_Robot.bLoadingReady AND NOT #in_Robot.bUnLoadingReady THEN
   //    #_iWorkStatus := #Status_Ready;
   //ELSIF #in_Robot.bLoadingReady AND NOT #in_Robot.bUnLoadingReady THEN
   //    #_iWorkStatus := #Status_Loading;
   //ELSIF NOT #in_Robot.bLoadingReady AND #in_Robot.bUnLoadingReady THEN
   //    #_iWorkStatus := #Status_UnLoading;
   //END_IF;
   //////////////////////////////////////////////////////////////////////////////////////////////

   /////////////////////////////////////////Логика работы////////////////////////////////////////
   //Статус: Готовности

   //Статус: Загрузка
       IF #_iWorkStatus = #Status_Loading THEN
       //ШАГ: Подготовка к Загрузке
       IF #_usiStepLoading = #Step_Ready THEN
           #_usiStepLoading := #Step_PreStart;
       END_IF;

       //ШАГ: Включаем вакуум
       IF (#tStepLoading[#Step_PreStart].ET > T#20ms AND #_usiCountTries = 0) THEN
           #_usiStepLoading := #Step_VacuumOn;
       END_IF;

       //ШАГ: Загрузка ОК
       IF  #_bSheetPressent THEN
           #_usiStepLoading := #Step_LoadingOk;
       END_IF;

       CASE #_usiStepLoading OF
           #Step_PreStart:
               //ШАГ: Подготовка к схватыванию
               #_bLoadingOK := FALSE;
               #_bUnLoadingOK := FALSE;
               #_usiCountTries := 0;

           #Step_VacuumOn:
               //ШАГ: Включаем вакуум
               #_Vacuum_bOn := TRUE;

           #Step_LoadingOk:
               //ШАГ: Загрузка ОК
               #_Vacuum_bOn := TRUE;
               #_bLoadingOK := TRUE;
       END_CASE;
   END_IF;

   //Статус: Разгрузка
   IF #_iWorkStatus = #Status_UnLoading THEN
       //ШАГ: Подготовка к разгрузке
       IF #_usiStepUnLoading = #Step_Ready
       THEN
           #_usiStepUnLoading := #Step_PreStart;
       END_IF;

       //ШАГ: Отключаем вакууум
       IF #tStepUnLoading[#Step_PreStart].ET > #cDelayUnloadVacuumOff THEN
           #_usiStepUnLoading := #Step_VacuumOn;
       END_IF;


       //ШАГ: Разгрузка ОК
       IF #tStepUnLoading[#Step_VacuumOn].ET > #cDelayUnloadVacuumOn THEN
           #_usiStepUnLoading := #Step_UnLoadingOk;
       END_IF;

       //ШАГ: В Автомате. Разгрузка
       CASE #_usiStepUnLoading OF
           #Step_PreStart:
               //ШАГ: Подготовка к разгрузке
               #_bLoadingOK := FALSE;
               #_bUnLoadingOK := FALSE;


           #Step_UnLoadingOk:
               //ШАГ: Разгрузка ОК
               #_bWaitingUnloading := FALSE;
               #_bUnLoadingOK := TRUE;
       END_CASE;
   ELSE
       #_usiStepUnLoading := #Step_Ready;
       #_bUnLoadingOK := FALSE;
   END_IF;
   //////////////////////////////////////////////////////////////////////////////////////////////

   //////////////////////////////////////////Доп. логика/////////////////////////////////////////
   //Счетчик попыток взятия листа
   #rtCountTries(CLK := #_usiStepLoading = #Step_VacuumOn);
   IF #rtCountTries.Q THEN
       #_usiCountTries := #_usiCountTries + 1;
   END_IF;
   //Бит готовности разгрузки
   IF #_bSheetPressent AND #_bLoadingOK THEN
       #_bWaitingUnloading := TRUE;
   END_IF;
   #tbWaitingUnloading(IN := #_A_bSheetLost OR #_A_bSheetTakeFail OR NOT #_bSheetPressent,
                    PT := T#1s);
   IF #tbWaitingUnloading.Q THEN
       #_bWaitingUnloading := FALSE;
   END_IF;
   //////////////////////////////////////////////////////////////////////////////////////////////

   ///////////////////////////////////////Выходные значения//////////////////////////////////////
   #rtVacuumOn(CLK := #_Vacuum_bOn);


   IF #rtVacuumOn.Q  THEN
       #_Vacuum_bOn := TRUE;
   END_IF;


   #out_A_bSheetTakeFail := #_A_bSheetTakeFail;
   #out_A_bSheetLost := #_A_bSheetLost;
   //#out_Robot.bLoadingOK := #_bLoadingOK;
   //#out_Robot.bUnloadingOK := #_bUnLoadingOK;
   //#out_Robot.bWaitingUnloading := #_bWaitingUnloading;
   //////////////////////////////////////////////////////////////////////////////////////////////

   ////////////////////////////////////////////Таймеры///////////////////////////////////////////
   //Запуск
   #tStepLoading[#_usiStepLoading](IN := TRUE,
                                   PT := T#1m);
   #tStepUnLoading[#_usiStepUnLoading](IN := TRUE,
                                     PT := T#1m);
   //Сброс
   FOR #i_tStepLoading := 0 TO 15 DO
       IF #_usiStepLoading <> #i_tStepLoading THEN
           #tStepLoading[#i_tStepLoading](IN := FALSE,
                                          PT := T#10s);
       END_IF;
   END_FOR;
   FOR #i_tStepUnLoading := 0 TO 15 DO
       IF #_usiStepUnLoading <> #i_tStepUnLoading THEN
           #tStepUnLoading[#i_tStepUnLoading](IN := FALSE,
                                              PT := T#10s);
       END_IF;
   END_FOR;
   ////////////////////////////////////////////////////////////////////////////////////////////// (156)
END_FUNCTION_BLOCK

FUNCTION_BLOCK "!Gripper"   // FB300, SCL
{ S7_Optimized_Access := 'TRUE' }
VERSION : 0.1
BEGIN
   //"!Gripper_DB"(in_Setting := "DataSetting".R1_Gripper,
   //                in_HMI_Control := "DataControl".R1_Gripper,
   //                in_IO := "DataIO".R1_InputGripper,
   //                in_Robot := "DataIO".R1_InputRobot,
   //                in_Sheet := NOT "InGripperGerconNC",
   //                in_usiCountTries:=0,
   //                in_bRobotExtControl:="From_KUKA1_EXT_ACTIVE",
   //                out_IO => "OutVacuumON",
   //                out_Robot => "SetVacuumON");
END_FUNCTION_BLOCK

// folder: 4_Working

